LIN {X 0,Y 474.699,Z 291.349,A -85,B 0,C 180,E1 -7395.456,E2 -7395.456} C_VEL
LIN {X 0,Y 474.663,Z 291.357,A -85,B 0,C 180,E1 -7399.01,E2 -7399.01} C_VEL
LIN {X 0,Y 474.587,Z 291.362,A -85,B 0,C 180,E1 -7401.729,E2 -7401.729} C_VEL
LIN {X 0,Y 474.657,Z 291.358,A -85,B 0,C 180,E1 -7404.493,E2 -7404.493} C_VEL
LIN {X 0,Y 474.68,Z 291.352,A -85,B 0,C 180,E1 -7407.334,E2 -7407.334} C_VEL
LIN {X 0,Y 474.603,Z 291.361,A -85,B 0,C 180,E1 -7410.23,E2 -7410.23} C_VEL
LIN {X 0,Y 474.641,Z 291.362,A -85,B 0,C 180,E1 -7413.22,E2 -7413.22} C_VEL
LIN {X 0,Y 474.587,Z 291.364,A -85,B 0,C 180,E1 -7416.324,E2 -7416.324} C_VEL
LIN {X 0,Y 474.617,Z 291.362,A -85,B 0,C 180,E1 -7419.646,E2 -7419.646} C_VEL
LIN {X 0,Y 474.614,Z 291.363,A -85,B 0,C 180,E1 -7422.934,E2 -7422.934} C_VEL
LIN {X 0,Y 474.604,Z 291.365,A -85,B 0,C 180,E1 -7425.895,E2 -7425.895} C_VEL
LIN {X 0,Y 474.627,Z 291.361,A -85,B 0,C 180,E1 -7429.041,E2 -7429.041} C_VEL
LIN {X 0,Y 474.61,Z 291.365,A -85,B 0,C 180,E1 -7431.704,E2 -7431.704} C_VEL
LIN {X 0,Y 474.624,Z 291.359,A -85,B 0,C 180,E1 -7434.726,E2 -7434.726} C_VEL
LIN {X 0,Y 474.636,Z 291.366,A -85,B 0,C 180,E1 -7437.788,E2 -7437.788} C_VEL
LIN {X 0,Y 474.641,Z 291.389,A -85,B 0,C 180,E1 -7439.43,E2 -7439.43} C_VEL
LIN {X 0,Y 475.664,Z 297.352,A -85,B 0,C 180,E1 -7440.661,E2 -7440.661} C_VEL
LIN {X 0,Y 475.45,Z 310.857,A -85,B 0,C 180,E1 -7443.24,E2 -7443.24} C_VEL
LIN {X 0,Y 478.358,Z 325.969,A -85,B 0,C 180,E1 -7443.591,E2 -7443.591} C_VEL
LIN {X 0,Y 477.959,Z 363.89,A -85,B 0,C 180,E1 -7444.164,E2 -7444.164} C_VEL
LIN {X 0,Y 477.193,Z 369.733,A -85,B 0,C 180,E1 -7444.225,E2 -7444.225} C_VEL
LIN {X 0,Y 471.606,Z 388.747,A -85,B 0,C 180,E1 -7444.31,E2 -7444.31} C_VEL
LIN {X 0,Y 470.888,Z 394.589,A -85,B 0,C 180,E1 -7444.374,E2 -7444.374} C_VEL
LIN {X 0,Y 470.679,Z 419.305,A -85,B 0,C 180,E1 -7444.785,E2 -7444.785} C_VEL
LIN {X 0,Y 470.335,Z 432.586,A -85,B 0,C 180,E1 -7445.178,E2 -7445.178} C_VEL
LIN {X 0,Y 470.093,Z 444.455,A -85,B 0,C 180,E1 -7445.702,E2 -7445.702} C_VEL
LIN {X 0,Y 469.632,Z 456.314,A -85,B 0,C 180,E1 -7446.402,E2 -7446.402} C_VEL
LIN {X 0,Y 469.071,Z 468.144,A -85,B 0,C 180,E1 -7447.306,E2 -7447.306} C_VEL
LIN {X 0,Y 468.611,Z 478.255,A -85,B 0,C 180,E1 -7448.276,E2 -7448.276} C_VEL
LIN {X 0,Y 468.134,Z 487.264,A -85,B 0,C 180,E1 -7449.341,E2 -7449.341} C_VEL
LIN {X 0,Y 467.759,Z 495.099,A -85,B 0,C 180,E1 -7450.47,E2 -7450.47} C_VEL
LIN {X 0,Y 467.356,Z 502.71,A -85,B 0,C 180,E1 -7451.818,E2 -7451.818} C_VEL
LIN {X 0,Y 467.119,Z 507.836,A -85,B 0,C 180,E1 -7452.939,E2 -7452.939} C_VEL
LIN {X 0,Y 466.914,Z 513.267,A -85,B 0,C 180,E1 -7454.436,E2 -7454.436} C_VEL
LIN {X 0,Y 466.804,Z 516.504,A -85,B 0,C 180,E1 -7455.616,E2 -7455.616} C_VEL
LIN {X 0,Y 466.642,Z 519.178,A -85,B 0,C 180,E1 -7456.943,E2 -7456.943} C_VEL
LIN {X 0,Y 466.683,Z 520.801,A -85,B 0,C 180,E1 -7458.2,E2 -7458.2} C_VEL
LIN {X 0,Y 466.618,Z 521.619,A -85,B 0,C 180,E1 -7459.587,E2 -7459.587} C_VEL
LIN {X 0,Y 466.608,Z 521.219,A -85,B 0,C 180,E1 -7461.337,E2 -7461.337} C_VEL
LIN {X 0,Y 466.648,Z 520.4,A -85,B 0,C 180,E1 -7462.209,E2 -7462.209} C_VEL
LIN {X 0,Y 466.771,Z 518.274,A -85,B 0,C 180,E1 -7463.585,E2 -7463.585} C_VEL
LIN {X 0,Y 466.796,Z 515.477,A -85,B 0,C 180,E1 -7464.817,E2 -7464.817} C_VEL
LIN {X 0,Y 466.926,Z 511.505,A -85,B 0,C 180,E1 -7466.116,E2 -7466.116} C_VEL
LIN {X 0,Y 467.112,Z 505.404,A -85,B 0,C 180,E1 -7467.628,E2 -7467.628} C_VEL
LIN {X 0,Y 467.432,Z 498.758,A -85,B 0,C 180,E1 -7468.923,E2 -7468.923} C_VEL
LIN {X 0,Y 467.848,Z 490.53,A -85,B 0,C 180,E1 -7470.215,E2 -7470.215} C_VEL
LIN {X 0,Y 468.168,Z 482.104,A -85,B 0,C 180,E1 -7471.29,E2 -7471.29} C_VEL
LIN {X 0,Y 468.605,Z 471.721,A -85,B 0,C 180,E1 -7472.363,E2 -7472.363} C_VEL
LIN {X 0,Y 469.234,Z 461.395,A -85,B 0,C 180,E1 -7473.219,E2 -7473.219} C_VEL
LIN {X 0,Y 469.692,Z 450.127,A -85,B 0,C 180,E1 -7473.968,E2 -7473.968} C_VEL
LIN {X 0,Y 470.052,Z 438.556,A -85,B 0,C 180,E1 -7474.555,E2 -7474.555} C_VEL
LIN {X 0,Y 470.323,Z 426.176,A -85,B 0,C 180,E1 -7475.009,E2 -7475.009} C_VEL
LIN {X 0,Y 470.539,Z 413.632,A -85,B 0,C 180,E1 -7475.302,E2 -7475.302} C_VEL
LIN {X 0,Y 471.218,Z 325.536,A -85,B 0,C 180,E1 -7476.65,E2 -7476.65} C_VEL
LIN {X 0,Y 468.385,Z 310.756,A -85,B 0,C 180,E1 -7477.002,E2 -7477.002} C_VEL
LIN {X 0,Y 468.608,Z 299.276,A -85,B 0,C 180,E1 -7479.277,E2 -7479.277} C_VEL
LIN {X 0,Y 467.603,Z 292.239,A -85,B 0,C 180,E1 -7480.746,E2 -7480.746} C_VEL
LIN {X 0,Y 467.583,Z 292.239,A -85,B 0,C 180,E1 -7483.029,E2 -7483.029} C_VEL
LIN {X 0,Y 467.623,Z 292.233,A -85,B 0,C 180,E1 -7485.873,E2 -7485.873} C_VEL
LIN {X 0,Y 467.615,Z 292.231,A -85,B 0,C 180,E1 -7489.307,E2 -7489.307} C_VEL
LIN {X 0,Y 467.529,Z 292.245,A -85,B 0,C 180,E1 -7492.073,E2 -7492.073} C_VEL
LIN {X 0,Y 467.551,Z 292.244,A -85,B 0,C 180,E1 -7494.889,E2 -7494.889} C_VEL
LIN {X 0,Y 467.542,Z 292.241,A -85,B 0,C 180,E1 -7497.773,E2 -7497.773} C_VEL
LIN {X 0,Y 467.543,Z 292.245,A -85,B 0,C 180,E1 -7501.04,E2 -7501.04} C_VEL
LIN {X 0,Y 467.573,Z 292.238,A -85,B 0,C 180,E1 -7504.239,E2 -7504.239} C_VEL
LIN {X 0,Y 467.542,Z 292.245,A -85,B 0,C 180,E1 -7507.185,E2 -7507.185} C_VEL
LIN {X 0,Y 467.553,Z 292.24,A -85,B 0,C 180,E1 -7510.266,E2 -7510.266} C_VEL
LIN {X 0,Y 467.54,Z 292.242,A -85,B 0,C 180,E1 -7513.745,E2 -7513.745} C_VEL
LIN {X 0,Y 467.541,Z 292.241,A -85,B 0,C 180,E1 -7516.254,E2 -7516.254} C_VEL
LIN {X 0,Y 467.568,Z 292.24,A -85,B 0,C 180,E1 -7518.723,E2 -7518.723} C_VEL
LIN {X 0,Y 467.556,Z 292.24,A -85,B 0,C 180,E1 -7521.955,E2 -7521.955} C_VEL
LIN {X 0,Y 467.557,Z 292.244,A -85,B 0,C 180,E1 -7525.167,E2 -7525.167} C_VEL
LIN {X 0,Y 467.575,Z 292.237,A -85,B 0,C 180,E1 -7528.259,E2 -7528.259} C_VEL
LIN {X 0,Y 467.565,Z 292.242,A -85,B 0,C 180,E1 -7531.25,E2 -7531.25} C_VEL
LIN {X 0,Y 467.583,Z 292.237,A -85,B 0,C 180,E1 -7534.158,E2 -7534.158} C_VEL
LIN {X 0,Y 467.567,Z 292.238,A -85,B 0,C 180,E1 -7536.995,E2 -7536.995} C_VEL
LIN {X 0,Y 467.614,Z 292.241,A -85,B 0,C 180,E1 -7539.777,E2 -7539.777} C_VEL
LIN {X 0,Y 467.599,Z 292.234,A -85,B 0,C 180,E1 -7542.506,E2 -7542.506} C_VEL
LIN {X 0,Y 467.596,Z 292.234,A -85,B 0,C 180,E1 -7545.196,E2 -7545.196} C_VEL
LIN {X 0,Y 467.647,Z 292.234,A -85,B 0,C 180,E1 -7547.854,E2 -7547.854} C_VEL
LIN {X 0,Y 467.672,Z 292.225,A -85,B 0,C 180,E1 -7551.357,E2 -7551.357} C_VEL
LIN {X 0,Y 467.712,Z 292.225,A -85,B 0,C 180,E1 -7553.962,E2 -7553.962} C_VEL
LIN {X 0,Y 467.85,Z 292.202,A -85,B 0,C 180,E1 -7557.417,E2 -7557.417} C_VEL
LIN {X 0,Y 467.871,Z 292.204,A -85,B 0,C 180,E1 -7560,E2 -7560} C_VEL
LIN {X 0,Y 467.85,Z 292.208,A -85,B 0,C 180,E1 -7562.583,E2 -7562.583} C_VEL
LIN {X 0,Y 467.734,Z 292.219,A -85,B 0,C 180,E1 -7566.038,E2 -7566.038} C_VEL
LIN {X 0,Y 467.674,Z 292.232,A -85,B 0,C 180,E1 -7568.643,E2 -7568.643} C_VEL
LIN {X 0,Y 467.648,Z 292.23,A -85,B 0,C 180,E1 -7572.146,E2 -7572.146} C_VEL
LIN {X 0,Y 467.631,Z 292.229,A -85,B 0,C 180,E1 -7575.695,E2 -7575.695} C_VEL
LIN {X 0,Y 467.609,Z 292.241,A -85,B 0,C 180,E1 -7578.765,E2 -7578.765} C_VEL
LIN {X 0,Y 467.572,Z 292.24,A -85,B 0,C 180,E1 -7581.269,E2 -7581.269} C_VEL
LIN {X 0,Y 467.566,Z 292.238,A -85,B 0,C 180,E1 -7583.944,E2 -7583.944} C_VEL
LIN {X 0,Y 467.621,Z 292.236,A -85,B 0,C 180,E1 -7586.8,E2 -7586.8} C_VEL
LIN {X 0,Y 467.582,Z 292.237,A -85,B 0,C 180,E1 -7589.736,E2 -7589.736} C_VEL
LIN {X 0,Y 467.577,Z 292.239,A -85,B 0,C 180,E1 -7592.759,E2 -7592.759} C_VEL
LIN {X 0,Y 467.55,Z 292.241,A -85,B 0,C 180,E1 -7595.89,E2 -7595.89} C_VEL
LIN {X 0,Y 467.577,Z 292.242,A -85,B 0,C 180,E1 -7599.145,E2 -7599.145} C_VEL
LIN {X 0,Y 467.582,Z 292.236,A -85,B 0,C 180,E1 -7602.568,E2 -7602.568} C_VEL
LIN {X 0,Y 467.566,Z 292.24,A -85,B 0,C 180,E1 -7605.054,E2 -7605.054} C_VEL
LIN {X 0,Y 467.585,Z 292.242,A -85,B 0,C 180,E1 -7607.441,E2 -7607.441} C_VEL
LIN {X 0,Y 467.557,Z 292.239,A -85,B 0,C 180,E1 -7610.854,E2 -7610.854} C_VEL
LIN {X 0,Y 467.557,Z 292.241,A -85,B 0,C 180,E1 -7614.262,E2 -7614.262} C_VEL
LIN {X 0,Y 467.58,Z 292.238,A -85,B 0,C 180,E1 -7617.322,E2 -7617.322} C_VEL
LIN {X 0,Y 467.569,Z 292.241,A -85,B 0,C 180,E1 -7620.668,E2 -7620.668} C_VEL
LIN {X 0,Y 467.628,Z 292.238,A -85,B 0,C 180,E1 -7623.683,E2 -7623.683} C_VEL
LIN {X 0,Y 467.684,Z 292.443,A -85,B 0,C 180,E1 -7624.106,E2 -7624.106} C_VEL
LIN {X 0,Y 469.76,Z 303.592,A -85,B 0,C 180,E1 -7626.176,E2 -7626.176} C_VEL
LIN {X 0,Y 469.177,Z 319.502,A -85,B 0,C 180,E1 -7628.931,E2 -7628.931} C_VEL
LIN {X 0,Y 468.445,Z 337.977,A -85,B 0,C 180,E1 -7632.089,E2 -7632.089} C_VEL
LIN {X 0,Y 468.223,Z 343.562,A -85,B 0,C 180,E1 -7633.037,E2 -7633.037} C_VEL
LIN {X 0,Y 471.029,Z 362.98,A -85,B 0,C 180,E1 -7633.437,E2 -7633.437} C_VEL
LIN {X 0,Y 470.381,Z 452.058,A -85,B 0,C 180,E1 -7634.816,E2 -7634.816} C_VEL
LIN {X 0,Y 470.087,Z 465.35,A -85,B 0,C 180,E1 -7635.194,E2 -7635.194} C_VEL
LIN {X 0,Y 469.635,Z 477.531,A -85,B 0,C 180,E1 -7635.705,E2 -7635.705} C_VEL
LIN {X 0,Y 469.193,Z 489.014,A -85,B 0,C 180,E1 -7636.355,E2 -7636.355} C_VEL
LIN {X 0,Y 468.662,Z 501.141,A -85,B 0,C 180,E1 -7637.25,E2 -7637.25} C_VEL
LIN {X 0,Y 468.214,Z 511.384,A -85,B 0,C 180,E1 -7638.2,E2 -7638.2} C_VEL
LIN {X 0,Y 467.766,Z 520.021,A -85,B 0,C 180,E1 -7639.176,E2 -7639.176} C_VEL
LIN {X 0,Y 467.411,Z 527.986,A -85,B 0,C 180,E1 -7640.262,E2 -7640.262} C_VEL
LIN {X 0,Y 467.109,Z 535.769,A -85,B 0,C 180,E1 -7641.565,E2 -7641.565} C_VEL
LIN {X 0,Y 466.85,Z 542.921,A -85,B 0,C 180,E1 -7643.083,E2 -7643.083} C_VEL
LIN {X 0,Y 466.76,Z 547.684,A -85,B 0,C 180,E1 -7644.384,E2 -7644.384} C_VEL
LIN {X 0,Y 466.647,Z 551.321,A -85,B 0,C 180,E1 -7645.682,E2 -7645.682} C_VEL
LIN {X 0,Y 466.69,Z 553.202,A -85,B 0,C 180,E1 -7646.547,E2 -7646.547} C_VEL
LIN {X 0,Y 466.662,Z 554.611,A -85,B 0,C 180,E1 -7647.411,E2 -7647.411} C_VEL
LIN {X 0,Y 466.619,Z 556.227,A -85,B 0,C 180,E1 -7649.137,E2 -7649.137} C_VEL
LIN {X 0,Y 466.601,Z 556.45,A -85,B 0,C 180,E1 -7650,E2 -7650} C_VEL
LIN {X 0,Y 466.619,Z 556.241,A -85,B 0,C 180,E1 -7650.863,E2 -7650.863} C_VEL
LIN {X 0,Y 466.662,Z 554.643,A -85,B 0,C 180,E1 -7652.59,E2 -7652.59} C_VEL
LIN {X 0,Y 466.69,Z 553.251,A -85,B 0,C 180,E1 -7653.454,E2 -7653.454} C_VEL
LIN {X 0,Y 466.689,Z 550.317,A -85,B 0,C 180,E1 -7654.751,E2 -7654.751} C_VEL
LIN {X 0,Y 466.751,Z 546.351,A -85,B 0,C 180,E1 -7656.051,E2 -7656.051} C_VEL
LIN {X 0,Y 466.943,Z 540.263,A -85,B 0,C 180,E1 -7657.568,E2 -7657.568} C_VEL
LIN {X 0,Y 467.186,Z 533.607,A -85,B 0,C 180,E1 -7658.87,E2 -7658.87} C_VEL
LIN {X 0,Y 467.537,Z 525.357,A -85,B 0,C 180,E1 -7660.174,E2 -7660.174} C_VEL
LIN {X 0,Y 468.026,Z 516.93,A -85,B 0,C 180,E1 -7661.257,E2 -7661.257} C_VEL
LIN {X 0,Y 468.529,Z 506.943,A -85,B 0,C 180,E1 -7662.305,E2 -7662.305} C_VEL
LIN {X 0,Y 468.957,Z 496.271,A -85,B 0,C 180,E1 -7663.212,E2 -7663.212} C_VEL
LIN {X 0,Y 469.489,Z 485.054,A -85,B 0,C 180,E1 -7663.968,E2 -7663.968} C_VEL
LIN {X 0,Y 469.977,Z 473.698,A -85,B 0,C 180,E1 -7664.561,E2 -7664.561} C_VEL
LIN {X 0,Y 470.38,Z 460.827,A -85,B 0,C 180,E1 -7665.047,E2 -7665.047} C_VEL
LIN {X 0,Y 470.681,Z 447.177,A -85,B 0,C 180,E1 -7665.369,E2 -7665.369} C_VEL
LIN {X 0,Y 471.268,Z 361.934,A -85,B 0,C 180,E1 -7666.688,E2 -7666.688} C_VEL
LIN {X 0,Y 468.32,Z 343.326,A -85,B 0,C 180,E1 -7667.112,E2 -7667.112} C_VEL
LIN {X 0,Y 469.089,Z 325.621,A -85,B 0,C 180,E1 -7670.157,E2 -7670.157} C_VEL
LIN {X 0,Y 469.915,Z 307.359,A -85,B 0,C 180,E1 -7673.349,E2 -7673.349} C_VEL
LIN {X 0,Y 469.787,Z 302.998,A -85,B 0,C 180,E1 -7674.138,E2 -7674.138} C_VEL
LIN {X 0,Y 467.646,Z 292.237,A -85,B 0,C 180,E1 -7676.257,E2 -7676.257} C_VEL
LIN {X 0,Y 467.572,Z 292.244,A -85,B 0,C 180,E1 -7679.332,E2 -7679.332} C_VEL
LIN {X 0,Y 467.584,Z 292.238,A -85,B 0,C 180,E1 -7682.679,E2 -7682.679} C_VEL
LIN {X 0,Y 467.561,Z 292.242,A -85,B 0,C 180,E1 -7685.739,E2 -7685.739} C_VEL
LIN {X 0,Y 467.561,Z 292.241,A -85,B 0,C 180,E1 -7689.147,E2 -7689.147} C_VEL
LIN {X 0,Y 467.588,Z 292.242,A -85,B 0,C 180,E1 -7692.567,E2 -7692.567} C_VEL
LIN {X 0,Y 467.566,Z 292.242,A -85,B 0,C 180,E1 -7695.052,E2 -7695.052} C_VEL
LIN {X 0,Y 467.59,Z 292.235,A -85,B 0,C 180,E1 -7697.44,E2 -7697.44} C_VEL
LIN {X 0,Y 467.576,Z 292.245,A -85,B 0,C 180,E1 -7700.854,E2 -7700.854} C_VEL
LIN {X 0,Y 467.559,Z 292.24,A -85,B 0,C 180,E1 -7704.261,E2 -7704.261} C_VEL
LIN {X 0,Y 467.581,Z 292.24,A -85,B 0,C 180,E1 -7707.321,E2 -7707.321} C_VEL
LIN {X 0,Y 467.569,Z 292.239,A -85,B 0,C 180,E1 -7710.667,E2 -7710.667} C_VEL
LIN {X 0,Y 467.615,Z 292.237,A -85,B 0,C 180,E1 -7713.199,E2 -7713.199} C_VEL
LIN {X 0,Y 467.592,Z 292.235,A -85,B 0,C 180,E1 -7716.468,E2 -7716.468} C_VEL
LIN {X 0,Y 467.621,Z 292.233,A -85,B 0,C 180,E1 -7719.777,E2 -7719.777} C_VEL
LIN {X 0,Y 467.607,Z 292.231,A -85,B 0,C 180,E1 -7722.507,E2 -7722.507} C_VEL
LIN {X 0,Y 467.608,Z 292.235,A -85,B 0,C 180,E1 -7725.196,E2 -7725.196} C_VEL
LIN {X 0,Y 467.654,Z 292.231,A -85,B 0,C 180,E1 -7727.854,E2 -7727.854} C_VEL
LIN {X 0,Y 467.68,Z 292.224,A -85,B 0,C 180,E1 -7731.357,E2 -7731.357} C_VEL
LIN {X 0,Y 467.741,Z 292.217,A -85,B 0,C 180,E1 -7733.962,E2 -7733.962} C_VEL
LIN {X 0,Y 467.858,Z 292.202,A -85,B 0,C 180,E1 -7737.417,E2 -7737.417} C_VEL
LIN {X 0,Y 467.88,Z 292.201,A -85,B 0,C 180,E1 -7740,E2 -7740} C_VEL
LIN {X 0,Y 467.857,Z 292.199,A -85,B 0,C 180,E1 -7742.583,E2 -7742.583} C_VEL
LIN {X 0,Y 467.732,Z 292.222,A -85,B 0,C 180,E1 -7746.037,E2 -7746.037} C_VEL
LIN {X 0,Y 467.679,Z 292.226,A -85,B 0,C 180,E1 -7748.643,E2 -7748.643} C_VEL
LIN {X 0,Y 467.654,Z 292.23,A -85,B 0,C 180,E1 -7752.145,E2 -7752.145} C_VEL
LIN {X 0,Y 467.638,Z 292.228,A -85,B 0,C 180,E1 -7755.695,E2 -7755.695} C_VEL
LIN {X 0,Y 467.616,Z 292.238,A -85,B 0,C 180,E1 -7758.764,E2 -7758.764} C_VEL
LIN {X 0,Y 467.579,Z 292.237,A -85,B 0,C 180,E1 -7761.268,E2 -7761.268} C_VEL
LIN {X 0,Y 467.571,Z 292.237,A -85,B 0,C 180,E1 -7763.943,E2 -7763.943} C_VEL
LIN {X 0,Y 467.616,Z 292.239,A -85,B 0,C 180,E1 -7766.8,E2 -7766.8} C_VEL
LIN {X 0,Y 467.552,Z 292.239,A -85,B 0,C 180,E1 -7769.738,E2 -7769.738} C_VEL
LIN {X 0,Y 467.582,Z 292.238,A -85,B 0,C 180,E1 -7772.758,E2 -7772.758} C_VEL
LIN {X 0,Y 467.552,Z 292.24,A -85,B 0,C 180,E1 -7775.89,E2 -7775.89} C_VEL
LIN {X 0,Y 467.575,Z 292.244,A -85,B 0,C 180,E1 -7779.145,E2 -7779.145} C_VEL
LIN {X 0,Y 467.586,Z 292.236,A -85,B 0,C 180,E1 -7782.567,E2 -7782.567} C_VEL
LIN {X 0,Y 467.565,Z 292.242,A -85,B 0,C 180,E1 -7785.053,E2 -7785.053} C_VEL
LIN {X 0,Y 467.589,Z 292.243,A -85,B 0,C 180,E1 -7787.44,E2 -7787.44} C_VEL
LIN {X 0,Y 467.56,Z 292.242,A -85,B 0,C 180,E1 -7790.853,E2 -7790.853} C_VEL
LIN {X 0,Y 467.56,Z 292.241,A -85,B 0,C 180,E1 -7794.261,E2 -7794.261} C_VEL
LIN {X 0,Y 467.582,Z 292.242,A -85,B 0,C 180,E1 -7797.321,E2 -7797.321} C_VEL
LIN {X 0,Y 467.594,Z 292.36,A -85,B 0,C 180,E1 -7799.239,E2 -7799.239} C_VEL
LIN {X 0,Y 468.745,Z 298.656,A -85,B 0,C 180,E1 -7800.557,E2 -7800.557} C_VEL
LIN {X 0,Y 468.479,Z 310.772,A -85,B 0,C 180,E1 -7802.933,E2 -7802.933} C_VEL
LIN {X 0,Y 471.552,Z 325.879,A -85,B 0,C 180,E1 -7803.319,E2 -7803.319} C_VEL
LIN {X 0,Y 470.888,Z 394.589,A -85,B 0,C 180,E1 -7804.374,E2 -7804.374} C_VEL
LIN {X 0,Y 470.185,Z 400.44,A -85,B 0,C 180,E1 -7804.435,E2 -7804.435} C_VEL
LIN {X 0,Y 464.632,Z 419.436,A -85,B 0,C 180,E1 -7804.553,E2 -7804.553} C_VEL
LIN {X 0,Y 463.798,Z 425.188,A -85,B 0,C 180,E1 -7804.679,E2 -7804.679} C_VEL
LIN {X 0,Y 463.444,Z 437.893,A -85,B 0,C 180,E1 -7805.138,E2 -7805.138} C_VEL
LIN {X 0,Y 463.017,Z 450.879,A -85,B 0,C 180,E1 -7805.806,E2 -7805.806} C_VEL
LIN {X 0,Y 462.522,Z 462.577,A -85,B 0,C 180,E1 -7806.611,E2 -7806.611} C_VEL
LIN {X 0,Y 461.987,Z 473.16,A -85,B 0,C 180,E1 -7807.529,E2 -7807.529} C_VEL
LIN {X 0,Y 461.451,Z 482.796,A -85,B 0,C 180,E1 -7808.56,E2 -7808.56} C_VEL
LIN {X 0,Y 460.975,Z 491.478,A -85,B 0,C 180,E1 -7809.705,E2 -7809.705} C_VEL
LIN {X 0,Y 460.513,Z 500.117,A -85,B 0,C 180,E1 -7811.12,E2 -7811.12} C_VEL
LIN {X 0,Y 460.2,Z 505.551,A -85,B 0,C 180,E1 -7812.216,E2 -7812.216} C_VEL
LIN {X 0,Y 459.96,Z 511.041,A -85,B 0,C 180,E1 -7813.58,E2 -7813.58} C_VEL
LIN {X 0,Y 459.776,Z 515.282,A -85,B 0,C 180,E1 -7814.938,E2 -7814.938} C_VEL
LIN {X 0,Y 459.663,Z 517.502,A -85,B 0,C 180,E1 -7815.84,E2 -7815.84} C_VEL
LIN {X 0,Y 459.579,Z 519.218,A -85,B 0,C 180,E1 -7816.739,E2 -7816.739} C_VEL
LIN {X 0,Y 459.589,Z 521.062,A -85,B 0,C 180,E1 -7818.148,E2 -7818.148} C_VEL
LIN {X 0,Y 459.537,Z 521.859,A -85,B 0,C 180,E1 -7819.425,E2 -7819.425} C_VEL
LIN {X 0,Y 459.504,Z 521.559,A -85,B 0,C 180,E1 -7821.202,E2 -7821.202} C_VEL
LIN {X 0,Y 459.543,Z 520.826,A -85,B 0,C 180,E1 -7822.088,E2 -7822.088} C_VEL
LIN {X 0,Y 459.694,Z 518.602,A -85,B 0,C 180,E1 -7823.589,E2 -7823.589} C_VEL
LIN {X 0,Y 459.7,Z 514.895,A -85,B 0,C 180,E1 -7825.176,E2 -7825.176} C_VEL
LIN {X 0,Y 459.897,Z 510.664,A -85,B 0,C 180,E1 -7826.495,E2 -7826.495} C_VEL
LIN {X 0,Y 460.144,Z 504.274,A -85,B 0,C 180,E1 -7828.03,E2 -7828.03} C_VEL
LIN {X 0,Y 460.532,Z 497.276,A -85,B 0,C 180,E1 -7829.344,E2 -7829.344} C_VEL
LIN {X 0,Y 460.953,Z 488.565,A -85,B 0,C 180,E1 -7830.655,E2 -7830.655} C_VEL
LIN {X 0,Y 461.333,Z 479.669,A -85,B 0,C 180,E1 -7831.745,E2 -7831.745} C_VEL
LIN {X 0,Y 461.819,Z 469.877,A -85,B 0,C 180,E1 -7832.725,E2 -7832.725} C_VEL
LIN {X 0,Y 462.457,Z 458.993,A -85,B 0,C 180,E1 -7833.594,E2 -7833.594} C_VEL
LIN {X 0,Y 462.878,Z 446.893,A -85,B 0,C 180,E1 -7834.353,E2 -7834.353} C_VEL
LIN {X 0,Y 463.252,Z 434.164,A -85,B 0,C 180,E1 -7834.949,E2 -7834.949} C_VEL
LIN {X 0,Y 463.548,Z 424.373,A -85,B 0,C 180,E1 -7835.273,E2 -7835.273} C_VEL
LIN {X 0,Y 463.692,Z 411.98,A -85,B 0,C 180,E1 -7835.544,E2 -7835.544} C_VEL
LIN {X 0,Y 464.345,Z 326.215,A -85,B 0,C 180,E1 -7836.873,E2 -7836.873} C_VEL
LIN {X 0,Y 461.404,Z 311.097,A -85,B 0,C 180,E1 -7837.218,E2 -7837.218} C_VEL
LIN {X 0,Y 461.623,Z 300.107,A -85,B 0,C 180,E1 -7839.419,E2 -7839.419} C_VEL
LIN {X 0,Y 460.573,Z 293.114,A -85,B 0,C 180,E1 -7840.912,E2 -7840.912} C_VEL
LIN {X 0,Y 460.537,Z 293.116,A -85,B 0,C 180,E1 -7843.232,E2 -7843.232} C_VEL
LIN {X 0,Y 460.578,Z 293.112,A -85,B 0,C 180,E1 -7845.987,E2 -7845.987} C_VEL
LIN {X 0,Y 460.562,Z 293.11,A -85,B 0,C 180,E1 -7849.615,E2 -7849.615} C_VEL
LIN {X 0,Y 460.505,Z 293.125,A -85,B 0,C 180,E1 -7852.428,E2 -7852.428} C_VEL
LIN {X 0,Y 460.529,Z 293.114,A -85,B 0,C 180,E1 -7855.792,E2 -7855.792} C_VEL
LIN {X 0,Y 460.516,Z 293.118,A -85,B 0,C 180,E1 -7859.232,E2 -7859.232} C_VEL
LIN {X 0,Y 460.525,Z 293.117,A -85,B 0,C 180,E1 -7862.284,E2 -7862.284} C_VEL
LIN {X 0,Y 460.504,Z 293.119,A -85,B 0,C 180,E1 -7865.445,E2 -7865.445} C_VEL
LIN {X 0,Y 460.524,Z 293.123,A -85,B 0,C 180,E1 -7868.894,E2 -7868.894} C_VEL
LIN {X 0,Y 460.485,Z 293.12,A -85,B 0,C 180,E1 -7872.184,E2 -7872.184} C_VEL
LIN {X 0,Y 460.506,Z 293.122,A -85,B 0,C 180,E1 -7875.41,E2 -7875.41} C_VEL
LIN {X 0,Y 460.52,Z 293.121,A -85,B 0,C 180,E1 -7878.988,E2 -7878.988} C_VEL
LIN {X 0,Y 460.508,Z 293.126,A -85,B 0,C 180,E1 -7881.265,E2 -7881.265} C_VEL
LIN {X 0,Y 460.503,Z 293.118,A -85,B 0,C 180,E1 -7884.554,E2 -7884.554} C_VEL
LIN {X 0,Y 460.523,Z 293.12,A -85,B 0,C 180,E1 -7887.715,E2 -7887.715} C_VEL
LIN {X 0,Y 460.529,Z 293.115,A -85,B 0,C 180,E1 -7890.768,E2 -7890.768} C_VEL
LIN {X 0,Y 460.537,Z 293.12,A -85,B 0,C 180,E1 -7893.733,E2 -7893.733} C_VEL
LIN {X 0,Y 460.536,Z 293.113,A -85,B 0,C 180,E1 -7896.623,E2 -7896.623} C_VEL
LIN {X 0,Y 460.542,Z 293.117,A -85,B 0,C 180,E1 -7899.452,E2 -7899.452} C_VEL
LIN {X 0,Y 460.55,Z 293.115,A -85,B 0,C 180,E1 -7902.23,E2 -7902.23} C_VEL
LIN {X 0,Y 460.559,Z 293.11,A -85,B 0,C 180,E1 -7904.965,E2 -7904.965} C_VEL
LIN {X 0,Y 460.602,Z 293.107,A -85,B 0,C 180,E1 -7908.559,E2 -7908.559} C_VEL
LIN {X 0,Y 460.657,Z 293.107,A -85,B 0,C 180,E1 -7912.108,E2 -7912.108} C_VEL
LIN {X 0,Y 460.681,Z 293.097,A -85,B 0,C 180,E1 -7914.748,E2 -7914.748} C_VEL
LIN {X 0,Y 460.792,Z 293.082,A -85,B 0,C 180,E1 -7917.378,E2 -7917.378} C_VEL
LIN {X 0,Y 460.842,Z 293.079,A -85,B 0,C 180,E1 -7920,E2 -7920} C_VEL
LIN {X 0,Y 460.791,Z 293.087,A -85,B 0,C 180,E1 -7922.623,E2 -7922.623} C_VEL
LIN {X 0,Y 460.701,Z 293.097,A -85,B 0,C 180,E1 -7926.13,E2 -7926.13} C_VEL
LIN {X 0,Y 460.621,Z 293.108,A -85,B 0,C 180,E1 -7928.776,E2 -7928.776} C_VEL
LIN {X 0,Y 460.605,Z 293.111,A -85,B 0,C 180,E1 -7932.445,E2 -7932.445} C_VEL
LIN {X 0,Y 460.592,Z 293.107,A -85,B 0,C 180,E1 -7935.998,E2 -7935.998} C_VEL
LIN {X 0,Y 460.563,Z 293.118,A -85,B 0,C 180,E1 -7938.902,E2 -7938.902} C_VEL
LIN {X 0,Y 460.508,Z 293.118,A -85,B 0,C 180,E1 -7941.486,E2 -7941.486} C_VEL
LIN {X 0,Y 460.535,Z 293.115,A -85,B 0,C 180,E1 -7944.333,E2 -7944.333} C_VEL
LIN {X 0,Y 460.578,Z 293.114,A -85,B 0,C 180,E1 -7947.244,E2 -7947.244} C_VEL
LIN {X 0,Y 460.524,Z 293.115,A -85,B 0,C 180,E1 -7950.239,E2 -7950.239} C_VEL
LIN {X 0,Y 460.523,Z 293.122,A -85,B 0,C 180,E1 -7953.326,E2 -7953.326} C_VEL
LIN {X 0,Y 460.473,Z 293.122,A -85,B 0,C 180,E1 -7956.53,E2 -7956.53} C_VEL
LIN {X 0,Y 460.553,Z 293.114,A -85,B 0,C 180,E1 -7959.86,E2 -7959.86} C_VEL
LIN {X 0,Y 460.512,Z 293.118,A -85,B 0,C 180,E1 -7962.902,E2 -7962.902} C_VEL
LIN {X 0,Y 460.507,Z 293.121,A -85,B 0,C 180,E1 -7965.831,E2 -7965.831} C_VEL
LIN {X 0,Y 460.527,Z 293.116,A -85,B 0,C 180,E1 -7968.99,E2 -7968.99} C_VEL
LIN {X 0,Y 460.515,Z 293.119,A -85,B 0,C 180,E1 -7971.267,E2 -7971.267} C_VEL
LIN {X 0,Y 460.508,Z 293.117,A -85,B 0,C 180,E1 -7974.555,E2 -7974.555} C_VEL
LIN {X 0,Y 460.53,Z 293.121,A -85,B 0,C 180,E1 -7977.717,E2 -7977.717} C_VEL
LIN {X 0,Y 460.539,Z 293.117,A -85,B 0,C 180,E1 -7980.77,E2 -7980.77} C_VEL
LIN {X 0,Y 460.608,Z 293.165,A -85,B 0,C 180,E1 -7983.897,E2 -7983.897} C_VEL
LIN {X 0,Y 462.732,Z 304.47,A -85,B 0,C 180,E1 -7986.03,E2 -7986.03} C_VEL
LIN {X 0,Y 462.372,Z 315.661,A -85,B 0,C 180,E1 -7988.002,E2 -7988.002} C_VEL
LIN {X 0,Y 461.625,Z 334.927,A -85,B 0,C 180,E1 -7991.355,E2 -7991.355} C_VEL
LIN {X 0,Y 461.209,Z 343.319,A -85,B 0,C 180,E1 -7992.801,E2 -7992.801} C_VEL
LIN {X 0,Y 464.194,Z 363.447,A -85,B 0,C 180,E1 -7993.22,E2 -7993.22} C_VEL
LIN {X 0,Y 463.482,Z 452.039,A -85,B 0,C 180,E1 -7994.612,E2 -7994.612} C_VEL
LIN {X 0,Y 463.152,Z 465.254,A -85,B 0,C 180,E1 -7994.995,E2 -7994.995} C_VEL
LIN {X 0,Y 462.698,Z 477.97,A -85,B 0,C 180,E1 -7995.543,E2 -7995.543} C_VEL
LIN {X 0,Y 462.182,Z 490.059,A -85,B 0,C 180,E1 -7996.256,E2 -7996.256} C_VEL
LIN {X 0,Y 461.659,Z 501.639,A -85,B 0,C 180,E1 -7997.14,E2 -7997.14} C_VEL
LIN {X 0,Y 461.178,Z 512.005,A -85,B 0,C 180,E1 -7998.128,E2 -7998.128} C_VEL
LIN {X 0,Y 460.665,Z 521.329,A -85,B 0,C 180,E1 -7999.229,E2 -7999.229} C_VEL
LIN {X 0,Y 460.227,Z 530.378,A -85,B 0,C 180,E1 -8000.552,E2 -8000.552} C_VEL
LIN {X 0,Y 459.941,Z 537.666,A -85,B 0,C 180,E1 -8001.875,E2 -8001.875} C_VEL
LIN {X 0,Y 459.727,Z 543.86,A -85,B 0,C 180,E1 -8003.295,E2 -8003.295} C_VEL
LIN {X 0,Y 459.65,Z 548.701,A -85,B 0,C 180,E1 -8004.737,E2 -8004.737} C_VEL
LIN {X 0,Y 459.564,Z 551.018,A -85,B 0,C 180,E1 -8005.615,E2 -8005.615} C_VEL
LIN {X 0,Y 459.586,Z 552.907,A -85,B 0,C 180,E1 -8006.494,E2 -8006.494} C_VEL
LIN {X 0,Y 459.584,Z 554.328,A -85,B 0,C 180,E1 -8007.371,E2 -8007.371} C_VEL
LIN {X 0,Y 459.552,Z 555.956,A -85,B 0,C 180,E1 -8009.124,E2 -8009.124} C_VEL
LIN {X 0,Y 459.532,Z 556.186,A -85,B 0,C 180,E1 -8010,E2 -8010} C_VEL
LIN {X 0,Y 459.523,Z 555.985,A -85,B 0,C 180,E1 -8010.877,E2 -8010.877} C_VEL
LIN {X 0,Y 459.584,Z 554.398,A -85,B 0,C 180,E1 -8012.63,E2 -8012.63} C_VEL
LIN {X 0,Y 459.585,Z 553.013,A -85,B 0,C 180,E1 -8013.507,E2 -8013.507} C_VEL
LIN {X 0,Y 459.617,Z 550.091,A -85,B 0,C 180,E1 -8014.825,E2 -8014.825} C_VEL
LIN {X 0,Y 459.715,Z 545.124,A -85,B 0,C 180,E1 -8016.431,E2 -8016.431} C_VEL
LIN {X 0,Y 459.903,Z 539.062,A -85,B 0,C 180,E1 -8017.905,E2 -8017.905} C_VEL
LIN {X 0,Y 460.187,Z 532.203,A -85,B 0,C 180,E1 -8019.228,E2 -8019.228} C_VEL
LIN {X 0,Y 460.588,Z 523.666,A -85,B 0,C 180,E1 -8020.551,E2 -8020.551} C_VEL
LIN {X 0,Y 461.113,Z 514.906,A -85,B 0,C 180,E1 -8021.651,E2 -8021.651} C_VEL
LIN {X 0,Y 461.689,Z 504.044,A -85,B 0,C 180,E1 -8022.761,E2 -8022.761} C_VEL
LIN {X 0,Y 462.184,Z 493.401,A -85,B 0,C 180,E1 -8023.633,E2 -8023.633} C_VEL
LIN {X 0,Y 462.757,Z 481.363,A -85,B 0,C 180,E1 -8024.4,E2 -8024.4} C_VEL
LIN {X 0,Y 463.308,Z 468.832,A -85,B 0,C 180,E1 -8025.001,E2 -8025.001} C_VEL
LIN {X 0,Y 463.699,Z 456.735,A -85,B 0,C 180,E1 -8025.409,E2 -8025.409} C_VEL
LIN {X 0,Y 463.973,Z 441.511,A -85,B 0,C 180,E1 -8025.71,E2 -8025.71} C_VEL
LIN {X 0,Y 464.561,Z 363.362,A -85,B 0,C 180,E1 -8026.934,E2 -8026.934} C_VEL
LIN {X 0,Y 461.375,Z 343.091,A -85,B 0,C 180,E1 -8027.398,E2 -8027.398} C_VEL
LIN {X 0,Y 462.172,Z 325.515,A -85,B 0,C 180,E1 -8030.472,E2 -8030.472} C_VEL
LIN {X 0,Y 463.001,Z 308.573,A -85,B 0,C 180,E1 -8033.482,E2 -8033.482} C_VEL
LIN {X 0,Y 462.79,Z 303.974,A -85,B 0,C 180,E1 -8034.332,E2 -8034.332} C_VEL
LIN {X 0,Y 460.593,Z 293.115,A -85,B 0,C 180,E1 -8036.508,E2 -8036.508} C_VEL
LIN {X 0,Y 460.533,Z 293.123,A -85,B 0,C 180,E1 -8039.558,E2 -8039.558} C_VEL
LIN {X 0,Y 460.533,Z 293.12,A -85,B 0,C 180,E1 -8042.284,E2 -8042.284} C_VEL
LIN {X 0,Y 460.512,Z 293.119,A -85,B 0,C 180,E1 -8045.445,E2 -8045.445} C_VEL
LIN {X 0,Y 460.535,Z 293.118,A -85,B 0,C 180,E1 -8048.896,E2 -8048.896} C_VEL
LIN {X 0,Y 460.524,Z 293.121,A -85,B 0,C 180,E1 -8052.181,E2 -8052.181} C_VEL
LIN {X 0,Y 460.514,Z 293.118,A -85,B 0,C 180,E1 -8055.411,E2 -8055.411} C_VEL
LIN {X 0,Y 460.532,Z 293.119,A -85,B 0,C 180,E1 -8058.397,E2 -8058.397} C_VEL
LIN {X 0,Y 460.523,Z 293.118,A -85,B 0,C 180,E1 -8061.266,E2 -8061.266} C_VEL
LIN {X 0,Y 460.51,Z 293.121,A -85,B 0,C 180,E1 -8064.554,E2 -8064.554} C_VEL
LIN {X 0,Y 460.531,Z 293.115,A -85,B 0,C 180,E1 -8067.715,E2 -8067.715} C_VEL
LIN {X 0,Y 460.539,Z 293.116,A -85,B 0,C 180,E1 -8070.769,E2 -8070.769} C_VEL
LIN {X 0,Y 460.558,Z 293.112,A -85,B 0,C 180,E1 -8073.734,E2 -8073.734} C_VEL
LIN {X 0,Y 460.545,Z 293.113,A -85,B 0,C 180,E1 -8076.624,E2 -8076.624} C_VEL
LIN {X 0,Y 460.551,Z 293.119,A -85,B 0,C 180,E1 -8079.453,E2 -8079.453} C_VEL
LIN {X 0,Y 460.558,Z 293.11,A -85,B 0,C 180,E1 -8082.23,E2 -8082.23} C_VEL
LIN {X 0,Y 460.566,Z 293.11,A -85,B 0,C 180,E1 -8084.965,E2 -8084.965} C_VEL
LIN {X 0,Y 460.609,Z 293.103,A -85,B 0,C 180,E1 -8088.559,E2 -8088.559} C_VEL
LIN {X 0,Y 460.694,Z 293.096,A -85,B 0,C 180,E1 -8092.108,E2 -8092.108} C_VEL
LIN {X 0,Y 460.694,Z 293.088,A -85,B 0,C 180,E1 -8094.748,E2 -8094.748} C_VEL
LIN {X 0,Y 460.799,Z 293.081,A -85,B 0,C 180,E1 -8097.377,E2 -8097.377} C_VEL
LIN {X 0,Y 460.85,Z 293.077,A -85,B 0,C 180,E1 -8100,E2 -8100} C_VEL
LIN {X 0,Y 460.798,Z 293.078,A -85,B 0,C 180,E1 -8102.622,E2 -8102.622} C_VEL
LIN {X 0,Y 460.699,Z 293.1,A -85,B 0,C 180,E1 -8106.13,E2 -8106.13} C_VEL
LIN {X 0,Y 460.626,Z 293.103,A -85,B 0,C 180,E1 -8108.776,E2 -8108.776} C_VEL
LIN {X 0,Y 460.612,Z 293.107,A -85,B 0,C 180,E1 -8112.445,E2 -8112.445} C_VEL
LIN {X 0,Y 460.599,Z 293.107,A -85,B 0,C 180,E1 -8115.998,E2 -8115.998} C_VEL
LIN {X 0,Y 460.569,Z 293.114,A -85,B 0,C 180,E1 -8118.902,E2 -8118.902} C_VEL
LIN {X 0,Y 460.514,Z 293.116,A -85,B 0,C 180,E1 -8121.486,E2 -8121.486} C_VEL
LIN {X 0,Y 460.541,Z 293.115,A -85,B 0,C 180,E1 -8124.332,E2 -8124.332} C_VEL
LIN {X 0,Y 460.572,Z 293.11,A -85,B 0,C 180,E1 -8127.244,E2 -8127.244} C_VEL
LIN {X 0,Y 460.509,Z 293.117,A -85,B 0,C 180,E1 -8130.24,E2 -8130.24} C_VEL
LIN {X 0,Y 460.528,Z 293.118,A -85,B 0,C 180,E1 -8133.325,E2 -8133.325} C_VEL
LIN {X 0,Y 460.475,Z 293.123,A -85,B 0,C 180,E1 -8136.53,E2 -8136.53} C_VEL
LIN {X 0,Y 460.526,Z 293.115,A -85,B 0,C 180,E1 -8139.863,E2 -8139.863} C_VEL
LIN {X 0,Y 460.512,Z 293.12,A -85,B 0,C 180,E1 -8142.9,E2 -8142.9} C_VEL
LIN {X 0,Y 460.506,Z 293.122,A -85,B 0,C 180,E1 -8145.831,E2 -8145.831} C_VEL
LIN {X 0,Y 460.53,Z 293.117,A -85,B 0,C 180,E1 -8148.989,E2 -8148.989} C_VEL
LIN {X 0,Y 460.519,Z 293.122,A -85,B 0,C 180,E1 -8151.266,E2 -8151.266} C_VEL
LIN {X 0,Y 460.51,Z 293.118,A -85,B 0,C 180,E1 -8154.554,E2 -8154.554} C_VEL
LIN {X 0,Y 460.533,Z 293.122,A -85,B 0,C 180,E1 -8157.716,E2 -8157.716} C_VEL
LIN {X 0,Y 460.541,Z 293.173,A -85,B 0,C 180,E1 -8159,E2 -8159} C_VEL
LIN {X 0,Y 461.833,Z 300.406,A -85,B 0,C 180,E1 -8160.534,E2 -8160.534} C_VEL
LIN {X 0,Y 461.587,Z 311.081,A -85,B 0,C 180,E1 -8162.653,E2 -8162.653} C_VEL
LIN {X 0,Y 464.85,Z 327.03,A -85,B 0,C 180,E1 -8163.058,E2 -8163.058} C_VEL
LIN {X 0,Y 463.919,Z 418.723,A -85,B 0,C 180,E1 -8164.511,E2 -8164.511} C_VEL
LIN {X 0,Y 463.798,Z 425.188,A -85,B 0,C 180,E1 -8164.679,E2 -8164.679} C_VEL
LIN {X 0,Y 462.337,Z 432.771,A -85,B 0,C 180,E1 -8164.881,E2 -8164.881} C_VEL
LIN {X 0,Y 459.73,Z 440.103,A -85,B 0,C 180,E1 -8165.093,E2 -8165.093} C_VEL
LIN {X 0,Y 456.85,Z 449.124,A -85,B 0,C 180,E1 -8165.465,E2 -8165.465} C_VEL
LIN {X 0,Y 456.093,Z 454.379,A -85,B 0,C 180,E1 -8165.769,E2 -8165.769} C_VEL
LIN {X 0,Y 455.524,Z 465.525,A -85,B 0,C 180,E1 -8166.592,E2 -8166.592} C_VEL
LIN {X 0,Y 454.904,Z 476.454,A -85,B 0,C 180,E1 -8167.618,E2 -8167.618} C_VEL
LIN {X 0,Y 454.357,Z 485.667,A -85,B 0,C 180,E1 -8168.685,E2 -8168.685} C_VEL
LIN {X 0,Y 453.9,Z 493.899,A -85,B 0,C 180,E1 -8169.848,E2 -8169.848} C_VEL
LIN {X 0,Y 453.399,Z 501.867,A -85,B 0,C 180,E1 -8171.238,E2 -8171.238} C_VEL
LIN {X 0,Y 453.119,Z 507.252,A -85,B 0,C 180,E1 -8172.395,E2 -8172.395} C_VEL
LIN {X 0,Y 452.849,Z 512.415,A -85,B 0,C 180,E1 -8173.778,E2 -8173.778} C_VEL
LIN {X 0,Y 452.681,Z 516.379,A -85,B 0,C 180,E1 -8175.157,E2 -8175.157} C_VEL
LIN {X 0,Y 452.502,Z 519.263,A -85,B 0,C 180,E1 -8176.528,E2 -8176.528} C_VEL
LIN {X 0,Y 452.512,Z 521.317,A -85,B 0,C 180,E1 -8178.086,E2 -8178.086} C_VEL
LIN {X 0,Y 452.446,Z 522.094,A -85,B 0,C 180,E1 -8179.257,E2 -8179.257} C_VEL
LIN {X 0,Y 452.416,Z 521.896,A -85,B 0,C 180,E1 -8181.063,E2 -8181.063} C_VEL
LIN {X 0,Y 452.456,Z 521.212,A -85,B 0,C 180,E1 -8181.964,E2 -8181.964} C_VEL
LIN {X 0,Y 452.603,Z 518.889,A -85,B 0,C 180,E1 -8183.611,E2 -8183.611} C_VEL
LIN {X 0,Y 452.625,Z 515.527,A -85,B 0,C 180,E1 -8185.101,E2 -8185.101} C_VEL
LIN {X 0,Y 452.817,Z 511.406,A -85,B 0,C 180,E1 -8186.44,E2 -8186.44} C_VEL
LIN {X 0,Y 453.078,Z 505.132,A -85,B 0,C 180,E1 -8187.999,E2 -8187.999} C_VEL
LIN {X 0,Y 453.438,Z 498.307,A -85,B 0,C 180,E1 -8189.333,E2 -8189.333} C_VEL
LIN {X 0,Y 453.916,Z 489.777,A -85,B 0,C 180,E1 -8190.665,E2 -8190.665} C_VEL
LIN {X 0,Y 454.277,Z 481.07,A -85,B 0,C 180,E1 -8191.773,E2 -8191.773} C_VEL
LIN {X 0,Y 454.753,Z 471.514,A -85,B 0,C 180,E1 -8192.768,E2 -8192.768} C_VEL
LIN {X 0,Y 455.428,Z 461.023,A -85,B 0,C 180,E1 -8193.649,E2 -8193.649} C_VEL
LIN {X 0,Y 455.897,Z 449.438,A -85,B 0,C 180,E1 -8194.42,E2 -8194.42} C_VEL
LIN {X 0,Y 456.344,Z 436.145,A -85,B 0,C 180,E1 -8195.08,E2 -8195.08} C_VEL
LIN {X 0,Y 456.563,Z 426.173,A -85,B 0,C 180,E1 -8195.437,E2 -8195.437} C_VEL
LIN {X 0,Y 456.8,Z 413.286,A -85,B 0,C 180,E1 -8195.739,E2 -8195.739} C_VEL
LIN {X 0,Y 457.588,Z 327.534,A -85,B 0,C 180,E1 -8197.085,E2 -8197.085} C_VEL
LIN {X 0,Y 454.454,Z 311.295,A -85,B 0,C 180,E1 -8197.466,E2 -8197.466} C_VEL
LIN {X 0,Y 454.632,Z 300.943,A -85,B 0,C 180,E1 -8199.565,E2 -8199.565} C_VEL
LIN {X 0,Y 453.566,Z 293.987,A -85,B 0,C 180,E1 -8201.054,E2 -8201.054} C_VEL
LIN {X 0,Y 453.499,Z 293.994,A -85,B 0,C 180,E1 -8203.441,E2 -8203.441} C_VEL
LIN {X 0,Y 453.536,Z 293.992,A -85,B 0,C 180,E1 -8206.196,E2 -8206.196} C_VEL
LIN {X 0,Y 453.515,Z 293.989,A -85,B 0,C 180,E1 -8209.038,E2 -8209.038} C_VEL
LIN {X 0,Y 453.474,Z 293.994,A -85,B 0,C 180,E1 -8211.835,E2 -8211.835} C_VEL
LIN {X 0,Y 453.464,Z 294.001,A -85,B 0,C 180,E1 -8214.736,E2 -8214.736} C_VEL
LIN {X 0,Y 453.459,Z 293.996,A -85,B 0,C 180,E1 -8217.942,E2 -8217.942} C_VEL
LIN {X 0,Y 453.461,Z 294.003,A -85,B 0,C 180,E1 -8220.76,E2 -8220.76} C_VEL
LIN {X 0,Y 453.464,Z 293.994,A -85,B 0,C 180,E1 -8223.913,E2 -8223.913} C_VEL
LIN {X 0,Y 453.447,Z 294.001,A -85,B 0,C 180,E1 -8227.189,E2 -8227.189} C_VEL
LIN {X 0,Y 453.465,Z 293.998,A -85,B 0,C 180,E1 -8230.611,E2 -8230.611} C_VEL
LIN {X 0,Y 453.453,Z 293.996,A -85,B 0,C 180,E1 -8234.221,E2 -8234.221} C_VEL
LIN {X 0,Y 453.442,Z 294.003,A -85,B 0,C 180,E1 -8237.003,E2 -8237.003} C_VEL
LIN {X 0,Y 453.487,Z 293.998,A -85,B 0,C 180,E1 -8239.409,E2 -8239.409} C_VEL
LIN {X 0,Y 453.444,Z 293.999,A -85,B 0,C 180,E1 -8242.81,E2 -8242.81} C_VEL
LIN {X 0,Y 453.469,Z 293.995,A -85,B 0,C 180,E1 -8246.087,E2 -8246.087} C_VEL
LIN {X 0,Y 453.468,Z 293.999,A -85,B 0,C 180,E1 -8249.24,E2 -8249.24} C_VEL
LIN {X 0,Y 453.524,Z 293.988,A -85,B 0,C 180,E1 -8252.297,E2 -8252.297} C_VEL
LIN {X 0,Y 453.491,Z 293.994,A -85,B 0,C 180,E1 -8255.264,E2 -8255.264} C_VEL
LIN {X 0,Y 453.472,Z 293.994,A -85,B 0,C 180,E1 -8258.415,E2 -8258.415} C_VEL
LIN {X 0,Y 453.513,Z 293.988,A -85,B 0,C 180,E1 -8261.008,E2 -8261.008} C_VEL
LIN {X 0,Y 453.568,Z 293.99,A -85,B 0,C 180,E1 -8263.876,E2 -8263.876} C_VEL
LIN {X 0,Y 453.555,Z 293.985,A -85,B 0,C 180,E1 -8267.471,E2 -8267.471} C_VEL
LIN {X 0,Y 453.583,Z 293.979,A -85,B 0,C 180,E1 -8271.087,E2 -8271.087} C_VEL
LIN {X 0,Y 453.642,Z 293.976,A -85,B 0,C 180,E1 -8273.774,E2 -8273.774} C_VEL
LIN {X 0,Y 453.736,Z 293.96,A -85,B 0,C 180,E1 -8277.337,E2 -8277.337} C_VEL
LIN {X 0,Y 453.812,Z 293.955,A -85,B 0,C 180,E1 -8280,E2 -8280} C_VEL
LIN {X 0,Y 453.735,Z 293.965,A -85,B 0,C 180,E1 -8282.663,E2 -8282.663} C_VEL
LIN {X 0,Y 453.668,Z 293.974,A -85,B 0,C 180,E1 -8286.226,E2 -8286.226} C_VEL
LIN {X 0,Y 453.585,Z 293.983,A -85,B 0,C 180,E1 -8288.914,E2 -8288.914} C_VEL
LIN {X 0,Y 453.555,Z 293.99,A -85,B 0,C 180,E1 -8292.529,E2 -8292.529} C_VEL
LIN {X 0,Y 453.537,Z 293.987,A -85,B 0,C 180,E1 -8296.196,E2 -8296.196} C_VEL
LIN {X 0,Y 453.512,Z 293.994,A -85,B 0,C 180,E1 -8299.041,E2 -8299.041} C_VEL
LIN {X 0,Y 453.469,Z 293.994,A -85,B 0,C 180,E1 -8301.837,E2 -8301.837} C_VEL
LIN {X 0,Y 453.507,Z 293.994,A -85,B 0,C 180,E1 -8304.735,E2 -8304.735} C_VEL
LIN {X 0,Y 453.532,Z 293.986,A -85,B 0,C 180,E1 -8307.962,E2 -8307.962} C_VEL
LIN {X 0,Y 453.478,Z 293.996,A -85,B 0,C 180,E1 -8310.76,E2 -8310.76} C_VEL
LIN {X 0,Y 453.471,Z 293.994,A -85,B 0,C 180,E1 -8313.913,E2 -8313.913} C_VEL
LIN {X 0,Y 453.465,Z 294.001,A -85,B 0,C 180,E1 -8317.189,E2 -8317.189} C_VEL
LIN {X 0,Y 453.512,Z 293.996,A -85,B 0,C 180,E1 -8319.448,E2 -8319.448} C_VEL
LIN {X 0,Y 453.464,Z 293.997,A -85,B 0,C 180,E1 -8322.995,E2 -8322.995} C_VEL
LIN {X 0,Y 453.462,Z 294,A -85,B 0,C 180,E1 -8325.78,E2 -8325.78} C_VEL
LIN {X 0,Y 453.475,Z 293.994,A -85,B 0,C 180,E1 -8328.21,E2 -8328.21} C_VEL
LIN {X 0,Y 453.484,Z 293.992,A -85,B 0,C 180,E1 -8330.795,E2 -8330.795} C_VEL
LIN {X 0,Y 453.452,Z 294.002,A -85,B 0,C 180,E1 -8333.918,E2 -8333.918} C_VEL
LIN {X 0,Y 453.481,Z 293.993,A -85,B 0,C 180,E1 -8337.152,E2 -8337.152} C_VEL
LIN {X 0,Y 453.474,Z 293.999,A -85,B 0,C 180,E1 -8340.269,E2 -8340.269} C_VEL
LIN {X 0,Y 453.538,Z 293.99,A -85,B 0,C 180,E1 -8343.297,E2 -8343.297} C_VEL
LIN {X 0,Y 453.6,Z 294.194,A -85,B 0,C 180,E1 -8343.742,E2 -8343.742} C_VEL
LIN {X 0,Y 455.766,Z 305.615,A -85,B 0,C 180,E1 -8345.933,E2 -8345.933} C_VEL
LIN {X 0,Y 455.423,Z 315.246,A -85,B 0,C 180,E1 -8347.655,E2 -8347.655} C_VEL
LIN {X 0,Y 454.739,Z 331.442,A -85,B 0,C 180,E1 -8350.52,E2 -8350.52} C_VEL
LIN {X 0,Y 454.222,Z 342.961,A -85,B 0,C 180,E1 -8352.539,E2 -8352.539} C_VEL
LIN {X 0,Y 457.334,Z 364.043,A -85,B 0,C 180,E1 -8353.001,E2 -8353.001} C_VEL
LIN {X 0,Y 456.6,Z 451.899,A -85,B 0,C 180,E1 -8354.403,E2 -8354.403} C_VEL
LIN {X 0,Y 456.258,Z 465.079,A -85,B 0,C 180,E1 -8354.792,E2 -8354.792} C_VEL
LIN {X 0,Y 455.786,Z 477.208,A -85,B 0,C 180,E1 -8355.318,E2 -8355.318} C_VEL
LIN {X 0,Y 455.227,Z 489.45,A -85,B 0,C 180,E1 -8356.042,E2 -8356.042} C_VEL
LIN {X 0,Y 454.672,Z 501.098,A -85,B 0,C 180,E1 -8356.939,E2 -8356.939} C_VEL
LIN {X 0,Y 454.179,Z 511.518,A -85,B 0,C 180,E1 -8357.943,E2 -8357.943} C_VEL
LIN {X 0,Y 453.658,Z 520.9,A -85,B 0,C 180,E1 -8359.061,E2 -8359.061} C_VEL
LIN {X 0,Y 453.188,Z 529.98,A -85,B 0,C 180,E1 -8360.404,E2 -8360.404} C_VEL
LIN {X 0,Y 452.869,Z 537.294,A -85,B 0,C 180,E1 -8361.747,E2 -8361.747} C_VEL
LIN {X 0,Y 452.69,Z 542.236,A -85,B 0,C 180,E1 -8362.866,E2 -8362.866} C_VEL
LIN {X 0,Y 452.554,Z 547.035,A -85,B 0,C 180,E1 -8364.207,E2 -8364.207} C_VEL
LIN {X 0,Y 452.486,Z 550.707,A -85,B 0,C 180,E1 -8365.546,E2 -8365.546} C_VEL
LIN {X 0,Y 452.484,Z 552.604,A -85,B 0,C 180,E1 -8366.439,E2 -8366.439} C_VEL
LIN {X 0,Y 452.508,Z 554.04,A -85,B 0,C 180,E1 -8367.33,E2 -8367.33} C_VEL
LIN {X 0,Y 452.457,Z 555.681,A -85,B 0,C 180,E1 -8369.11,E2 -8369.11} C_VEL
LIN {X 0,Y 452.465,Z 555.92,A -85,B 0,C 180,E1 -8370,E2 -8370} C_VEL
LIN {X 0,Y 452.43,Z 555.731,A -85,B 0,C 180,E1 -8370.891,E2 -8370.891} C_VEL
LIN {X 0,Y 452.508,Z 554.158,A -85,B 0,C 180,E1 -8372.671,E2 -8372.671} C_VEL
LIN {X 0,Y 452.482,Z 552.78,A -85,B 0,C 180,E1 -8373.562,E2 -8373.562} C_VEL
LIN {X 0,Y 452.545,Z 549.873,A -85,B 0,C 180,E1 -8374.9,E2 -8374.9} C_VEL
LIN {X 0,Y 452.611,Z 545.424,A -85,B 0,C 180,E1 -8376.396,E2 -8376.396} C_VEL
LIN {X 0,Y 452.779,Z 540.877,A -85,B 0,C 180,E1 -8377.582,E2 -8377.582} C_VEL
LIN {X 0,Y 453.054,Z 534.527,A -85,B 0,C 180,E1 -8378.924,E2 -8378.924} C_VEL
LIN {X 0,Y 453.42,Z 526.592,A -85,B 0,C 180,E1 -8380.268,E2 -8380.268} C_VEL
LIN {X 0,Y 453.95,Z 518.528,A -85,B 0,C 180,E1 -8381.385,E2 -8381.385} C_VEL
LIN {X 0,Y 454.497,Z 508.705,A -85,B 0,C 180,E1 -8382.503,E2 -8382.503} C_VEL
LIN {X 0,Y 455.069,Z 497.749,A -85,B 0,C 180,E1 -8383.509,E2 -8383.509} C_VEL
LIN {X 0,Y 455.715,Z 485.266,A -85,B 0,C 180,E1 -8384.4,E2 -8384.4} C_VEL
LIN {X 0,Y 456.346,Z 473.003,A -85,B 0,C 180,E1 -8385.064,E2 -8385.064} C_VEL
LIN {X 0,Y 456.816,Z 460.063,A -85,B 0,C 180,E1 -8385.562,E2 -8385.562} C_VEL
LIN {X 0,Y 457.124,Z 446.297,A -85,B 0,C 180,E1 -8385.894,E2 -8385.894} C_VEL
LIN {X 0,Y 457.848,Z 364.68,A -85,B 0,C 180,E1 -8387.193,E2 -8387.193} C_VEL
LIN {X 0,Y 454.699,Z 344.39,A -85,B 0,C 180,E1 -8387.661,E2 -8387.661} C_VEL
LIN {X 0,Y 454.443,Z 342.809,A -85,B 0,C 180,E1 -8387.703,E2 -8387.703} C_VEL
LIN {X 0,Y 455.293,Z 325.423,A -85,B 0,C 180,E1 -8390.796,E2 -8390.796} C_VEL
LIN {X 0,Y 456.193,Z 308.523,A -85,B 0,C 180,E1 -8393.849,E2 -8393.849} C_VEL
LIN {X 0,Y 455.211,Z 301.979,A -85,B 0,C 180,E1 -8395.124,E2 -8395.124} C_VEL
LIN {X 0,Y 453.564,Z 293.991,A -85,B 0,C 180,E1 -8396.765,E2 -8396.765} C_VEL
LIN {X 0,Y 453.475,Z 294.005,A -85,B 0,C 180,E1 -8399.785,E2 -8399.785} C_VEL
LIN {X 0,Y 453.492,Z 293.992,A -85,B 0,C 180,E1 -8403.189,E2 -8403.189} C_VEL
LIN {X 0,Y 453.455,Z 294.004,A -85,B 0,C 180,E1 -8406.299,E2 -8406.299} C_VEL
LIN {X 0,Y 453.484,Z 293.994,A -85,B 0,C 180,E1 -8409.45,E2 -8409.45} C_VEL
LIN {X 0,Y 453.477,Z 293.996,A -85,B 0,C 180,E1 -8411.935,E2 -8411.935} C_VEL
LIN {X 0,Y 453.485,Z 293.994,A -85,B 0,C 180,E1 -8415.471,E2 -8415.471} C_VEL
LIN {X 0,Y 453.479,Z 293.995,A -85,B 0,C 180,E1 -8418.209,E2 -8418.209} C_VEL
LIN {X 0,Y 453.491,Z 293.998,A -85,B 0,C 180,E1 -8420.794,E2 -8420.794} C_VEL
LIN {X 0,Y 453.454,Z 293.996,A -85,B 0,C 180,E1 -8423.917,E2 -8423.917} C_VEL
LIN {X 0,Y 453.482,Z 293.999,A -85,B 0,C 180,E1 -8427.151,E2 -8427.151} C_VEL
LIN {X 0,Y 453.474,Z 293.992,A -85,B 0,C 180,E1 -8430.268,E2 -8430.268} C_VEL
LIN {X 0,Y 453.504,Z 293.994,A -85,B 0,C 180,E1 -8433.294,E2 -8433.294} C_VEL
LIN {X 0,Y 453.501,Z 293.99,A -85,B 0,C 180,E1 -8436.239,E2 -8436.239} C_VEL
LIN {X 0,Y 453.482,Z 293.997,A -85,B 0,C 180,E1 -8439.117,E2 -8439.117} C_VEL
LIN {X 0,Y 453.51,Z 293.99,A -85,B 0,C 180,E1 -8441.944,E2 -8441.944} C_VEL
LIN {X 0,Y 453.54,Z 293.984,A -85,B 0,C 180,E1 -8444.726,E2 -8444.726} C_VEL
LIN {X 0,Y 453.558,Z 293.982,A -85,B 0,C 180,E1 -8448.379,E2 -8448.379} C_VEL
LIN {X 0,Y 453.651,Z 293.975,A -85,B 0,C 180,E1 -8451.985,E2 -8451.985} C_VEL
LIN {X 0,Y 453.668,Z 293.964,A -85,B 0,C 180,E1 -8454.667,E2 -8454.667} C_VEL
LIN {X 0,Y 453.743,Z 293.959,A -85,B 0,C 180,E1 -8457.337,E2 -8457.337} C_VEL
LIN {X 0,Y 453.821,Z 293.952,A -85,B 0,C 180,E1 -8460,E2 -8460} C_VEL
LIN {X 0,Y 453.742,Z 293.956,A -85,B 0,C 180,E1 -8462.663,E2 -8462.663} C_VEL
LIN {X 0,Y 453.667,Z 293.974,A -85,B 0,C 180,E1 -8466.225,E2 -8466.225} C_VEL
LIN {X 0,Y 453.59,Z 293.979,A -85,B 0,C 180,E1 -8468.913,E2 -8468.913} C_VEL
LIN {X 0,Y 453.562,Z 293.986,A -85,B 0,C 180,E1 -8472.529,E2 -8472.529} C_VEL
LIN {X 0,Y 453.543,Z 293.988,A -85,B 0,C 180,E1 -8476.196,E2 -8476.196} C_VEL
LIN {X 0,Y 453.518,Z 293.991,A -85,B 0,C 180,E1 -8479.041,E2 -8479.041} C_VEL
LIN {X 0,Y 453.475,Z 293.993,A -85,B 0,C 180,E1 -8481.836,E2 -8481.836} C_VEL
LIN {X 0,Y 453.513,Z 293.992,A -85,B 0,C 180,E1 -8484.734,E2 -8484.734} C_VEL
LIN {X 0,Y 453.531,Z 293.983,A -85,B 0,C 180,E1 -8487.96,E2 -8487.96} C_VEL
LIN {X 0,Y 453.464,Z 293.994,A -85,B 0,C 180,E1 -8491.525,E2 -8491.525} C_VEL
LIN {X 0,Y 453.486,Z 293.995,A -85,B 0,C 180,E1 -8494.777,E2 -8494.777} C_VEL
LIN {X 0,Y 453.462,Z 293.995,A -85,B 0,C 180,E1 -8498.312,E2 -8498.312} C_VEL
LIN {X 0,Y 453.493,Z 293.99,A -85,B 0,C 180,E1 -8500.609,E2 -8500.609} C_VEL
LIN {X 0,Y 453.454,Z 294.002,A -85,B 0,C 180,E1 -8503.244,E2 -8503.244} C_VEL
LIN {X 0,Y 453.461,Z 294,A -85,B 0,C 180,E1 -8505.779,E2 -8505.779} C_VEL
LIN {X 0,Y 453.479,Z 293.994,A -85,B 0,C 180,E1 -8508.209,E2 -8508.209} C_VEL
LIN {X 0,Y 453.487,Z 293.995,A -85,B 0,C 180,E1 -8510.795,E2 -8510.795} C_VEL
LIN {X 0,Y 453.454,Z 294.001,A -85,B 0,C 180,E1 -8513.917,E2 -8513.917} C_VEL
LIN {X 0,Y 453.484,Z 293.998,A -85,B 0,C 180,E1 -8517.151,E2 -8517.151} C_VEL
LIN {X 0,Y 453.516,Z 294.144,A -85,B 0,C 180,E1 -8518.782,E2 -8518.782} C_VEL
LIN {X 0,Y 454.904,Z 301.506,A -85,B 0,C 180,E1 -8520.371,E2 -8520.371} C_VEL
LIN {X 0,Y 454.684,Z 311.398,A -85,B 0,C 180,E1 -8522.356,E2 -8522.356} C_VEL
LIN {X 0,Y 458.125,Z 327.942,A -85,B 0,C 180,E1 -8522.783,E2 -8522.783} C_VEL
LIN {X 0,Y 457.193,Z 418.249,A -85,B 0,C 180,E1 -8524.231,E2 -8524.231} C_VEL
LIN {X 0,Y 456.83,Z 431.271,A -85,B 0,C 180,E1 -8524.606,E2 -8524.606} C_VEL
LIN {X 0,Y 456.525,Z 443.811,A -85,B 0,C 180,E1 -8525.155,E2 -8525.155} C_VEL
LIN {X 0,Y 456.093,Z 454.379,A -85,B 0,C 180,E1 -8525.769,E2 -8525.769} C_VEL
LIN {X 0,Y 455.226,Z 459.607,A -85,B 0,C 180,E1 -8526.1,E2 -8526.1} C_VEL
LIN {X 0,Y 451.977,Z 467.901,A -85,B 0,C 180,E1 -8526.656,E2 -8526.656} C_VEL
LIN {X 0,Y 448.712,Z 475.73,A -85,B 0,C 180,E1 -8527.306,E2 -8527.306} C_VEL
LIN {X 0,Y 447.823,Z 480.221,A -85,B 0,C 180,E1 -8527.78,E2 -8527.78} C_VEL
LIN {X 0,Y 447.18,Z 490.126,A -85,B 0,C 180,E1 -8529.05,E2 -8529.05} C_VEL
LIN {X 0,Y 446.752,Z 497.603,A -85,B 0,C 180,E1 -8530.231,E2 -8530.231} C_VEL
LIN {X 0,Y 446.243,Z 504.871,A -85,B 0,C 180,E1 -8531.64,E2 -8531.64} C_VEL
LIN {X 0,Y 445.906,Z 510.602,A -85,B 0,C 180,E1 -8533.047,E2 -8533.047} C_VEL
LIN {X 0,Y 445.689,Z 515.067,A -85,B 0,C 180,E1 -8534.45,E2 -8534.45} C_VEL
LIN {X 0,Y 445.585,Z 517.41,A -85,B 0,C 180,E1 -8535.382,E2 -8535.382} C_VEL
LIN {X 0,Y 445.447,Z 519.304,A -85,B 0,C 180,E1 -8536.31,E2 -8536.31} C_VEL
LIN {X 0,Y 445.428,Z 521.58,A -85,B 0,C 180,E1 -8538.026,E2 -8538.026} C_VEL
LIN {X 0,Y 445.356,Z 522.295,A -85,B 0,C 180,E1 -8539.084,E2 -8539.084} C_VEL
LIN {X 0,Y 445.309,Z 522.482,A -85,B 0,C 180,E1 -8540.002,E2 -8540.002} C_VEL
LIN {X 0,Y 445.351,Z 521.596,A -85,B 0,C 180,E1 -8541.834,E2 -8541.834} C_VEL
LIN {X 0,Y 445.442,Z 520.569,A -85,B 0,C 180,E1 -8542.748,E2 -8542.748} C_VEL
LIN {X 0,Y 445.529,Z 519.118,A -85,B 0,C 180,E1 -8543.66,E2 -8543.66} C_VEL
LIN {X 0,Y 445.553,Z 516.151,A -85,B 0,C 180,E1 -8545.023,E2 -8545.023} C_VEL
LIN {X 0,Y 445.74,Z 512.136,A -85,B 0,C 180,E1 -8546.384,E2 -8546.384} C_VEL
LIN {X 0,Y 446.006,Z 505.977,A -85,B 0,C 180,E1 -8547.968,E2 -8547.968} C_VEL
LIN {X 0,Y 446.351,Z 499.282,A -85,B 0,C 180,E1 -8549.323,E2 -8549.323} C_VEL
LIN {X 0,Y 446.852,Z 490.972,A -85,B 0,C 180,E1 -8550.675,E2 -8550.675} C_VEL
LIN {X 0,Y 447.226,Z 482.448,A -85,B 0,C 180,E1 -8551.801,E2 -8551.801} C_VEL
LIN {X 0,Y 447.775,Z 471.952,A -85,B 0,C 180,E1 -8552.923,E2 -8552.923} C_VEL
LIN {X 0,Y 448.49,Z 461.491,A -85,B 0,C 180,E1 -8553.818,E2 -8553.818} C_VEL
LIN {X 0,Y 448.982,Z 449.981,A -85,B 0,C 180,E1 -8554.601,E2 -8554.601} C_VEL
LIN {X 0,Y 449.416,Z 438.047,A -85,B 0,C 180,E1 -8555.215,E2 -8555.215} C_VEL
LIN {X 0,Y 449.619,Z 426.974,A -85,B 0,C 180,E1 -8555.634,E2 -8555.634} C_VEL
LIN {X 0,Y 449.921,Z 414.371,A -85,B 0,C 180,E1 -8555.939,E2 -8555.939} C_VEL
LIN {X 0,Y 450.65,Z 327.848,A -85,B 0,C 180,E1 -8557.323,E2 -8557.323} C_VEL
LIN {X 0,Y 447.499,Z 311.476,A -85,B 0,C 180,E1 -8557.724,E2 -8557.724} C_VEL
LIN {X 0,Y 447.645,Z 301.774,A -85,B 0,C 180,E1 -8559.716,E2 -8559.716} C_VEL
LIN {X 0,Y 446.496,Z 294.868,A -85,B 0,C 180,E1 -8561.232,E2 -8561.232} C_VEL
LIN {X 0,Y 446.459,Z 294.872,A -85,B 0,C 180,E1 -8563.657,E2 -8563.657} C_VEL
LIN {X 0,Y 446.483,Z 294.871,A -85,B 0,C 180,E1 -8566.459,E2 -8566.459} C_VEL
LIN {X 0,Y 446.466,Z 294.866,A -85,B 0,C 180,E1 -8569.303,E2 -8569.303} C_VEL
LIN {X 0,Y 446.415,Z 294.877,A -85,B 0,C 180,E1 -8572.199,E2 -8572.199} C_VEL
LIN {X 0,Y 446.416,Z 294.874,A -85,B 0,C 180,E1 -8575.154,E2 -8575.154} C_VEL
LIN {X 0,Y 446.433,Z 294.873,A -85,B 0,C 180,E1 -8578.181,E2 -8578.181} C_VEL
LIN {X 0,Y 446.408,Z 294.875,A -85,B 0,C 180,E1 -8581.3,E2 -8581.3} C_VEL
LIN {X 0,Y 446.419,Z 294.876,A -85,B 0,C 180,E1 -8584.523,E2 -8584.523} C_VEL
LIN {X 0,Y 446.407,Z 294.874,A -85,B 0,C 180,E1 -8588.078,E2 -8588.078} C_VEL
LIN {X 0,Y 446.4,Z 294.878,A -85,B 0,C 180,E1 -8591.393,E2 -8591.393} C_VEL
LIN {X 0,Y 446.444,Z 294.878,A -85,B 0,C 180,E1 -8595.103,E2 -8595.103} C_VEL
LIN {X 0,Y 446.412,Z 294.874,A -85,B 0,C 180,E1 -8598.607,E2 -8598.607} C_VEL
LIN {X 0,Y 446.405,Z 294.875,A -85,B 0,C 180,E1 -8601.921,E2 -8601.921} C_VEL
LIN {X 0,Y 446.422,Z 294.879,A -85,B 0,C 180,E1 -8605.476,E2 -8605.476} C_VEL
LIN {X 0,Y 446.408,Z 294.874,A -85,B 0,C 180,E1 -8608.699,E2 -8608.699} C_VEL
LIN {X 0,Y 446.477,Z 294.87,A -85,B 0,C 180,E1 -8611.821,E2 -8611.821} C_VEL
LIN {X 0,Y 446.434,Z 294.87,A -85,B 0,C 180,E1 -8614.846,E2 -8614.846} C_VEL
LIN {X 0,Y 446.44,Z 294.871,A -85,B 0,C 180,E1 -8618.245,E2 -8618.245} C_VEL
LIN {X 0,Y 446.449,Z 294.874,A -85,B 0,C 180,E1 -8621.649,E2 -8621.649} C_VEL
LIN {X 0,Y 446.507,Z 294.862,A -85,B 0,C 180,E1 -8624.48,E2 -8624.48} C_VEL
LIN {X 0,Y 446.509,Z 294.867,A -85,B 0,C 180,E1 -8628.193,E2 -8628.193} C_VEL
LIN {X 0,Y 446.529,Z 294.858,A -85,B 0,C 180,E1 -8630.945,E2 -8630.945} C_VEL
LIN {X 0,Y 446.61,Z 294.851,A -85,B 0,C 180,E1 -8633.676,E2 -8633.676} C_VEL
LIN {X 0,Y 446.683,Z 294.839,A -85,B 0,C 180,E1 -8637.295,E2 -8637.295} C_VEL
LIN {X 0,Y 446.782,Z 294.831,A -85,B 0,C 180,E1 -8640,E2 -8640} C_VEL
LIN {X 0,Y 446.682,Z 294.843,A -85,B 0,C 180,E1 -8642.706,E2 -8642.706} C_VEL
LIN {X 0,Y 446.638,Z 294.851,A -85,B 0,C 180,E1 -8646.324,E2 -8646.324} C_VEL
LIN {X 0,Y 446.531,Z 294.86,A -85,B 0,C 180,E1 -8649.056,E2 -8649.056} C_VEL
LIN {X 0,Y 446.513,Z 294.868,A -85,B 0,C 180,E1 -8652.73,E2 -8652.73} C_VEL
LIN {X 0,Y 446.488,Z 294.865,A -85,B 0,C 180,E1 -8656.228,E2 -8656.228} C_VEL
LIN {X 0,Y 446.461,Z 294.869,A -85,B 0,C 180,E1 -8659.304,E2 -8659.304} C_VEL
LIN {X 0,Y 446.41,Z 294.874,A -85,B 0,C 180,E1 -8662.2,E2 -8662.2} C_VEL
LIN {X 0,Y 446.452,Z 294.874,A -85,B 0,C 180,E1 -8665.153,E2 -8665.153} C_VEL
LIN {X 0,Y 446.478,Z 294.865,A -85,B 0,C 180,E1 -8668.179,E2 -8668.179} C_VEL
LIN {X 0,Y 446.428,Z 294.877,A -85,B 0,C 180,E1 -8671.3,E2 -8671.3} C_VEL
LIN {X 0,Y 446.424,Z 294.872,A -85,B 0,C 180,E1 -8674.524,E2 -8674.524} C_VEL
LIN {X 0,Y 446.425,Z 294.872,A -85,B 0,C 180,E1 -8678.083,E2 -8678.083} C_VEL
LIN {X 0,Y 446.423,Z 294.874,A -85,B 0,C 180,E1 -8680.919,E2 -8680.919} C_VEL
LIN {X 0,Y 446.419,Z 294.876,A -85,B 0,C 180,E1 -8683.844,E2 -8683.844} C_VEL
LIN {X 0,Y 446.395,Z 294.875,A -85,B 0,C 180,E1 -8686.404,E2 -8686.404} C_VEL
LIN {X 0,Y 446.423,Z 294.873,A -85,B 0,C 180,E1 -8689.083,E2 -8689.083} C_VEL
LIN {X 0,Y 446.404,Z 294.877,A -85,B 0,C 180,E1 -8692.122,E2 -8692.122} C_VEL
LIN {X 0,Y 446.427,Z 294.875,A -85,B 0,C 180,E1 -8695.478,E2 -8695.478} C_VEL
LIN {X 0,Y 446.414,Z 294.873,A -85,B 0,C 180,E1 -8698.701,E2 -8698.701} C_VEL
LIN {X 0,Y 446.484,Z 294.871,A -85,B 0,C 180,E1 -8701.822,E2 -8701.822} C_VEL
LIN {X 0,Y 446.527,Z 294.901,A -85,B 0,C 180,E1 -8703.523,E2 -8703.523} C_VEL
LIN {X 0,Y 448.864,Z 307.535,A -85,B 0,C 180,E1 -8705.979,E2 -8705.979} C_VEL
LIN {X 0,Y 448.102,Z 324.791,A -85,B 0,C 180,E1 -8709.096,E2 -8709.096} C_VEL
LIN {X 0,Y 447.267,Z 342.667,A -85,B 0,C 180,E1 -8712.285,E2 -8712.285} C_VEL
LIN {X 0,Y 450.494,Z 365.199,A -85,B 0,C 180,E1 -8712.788,E2 -8712.788} C_VEL
LIN {X 0,Y 449.715,Z 451.646,A -85,B 0,C 180,E1 -8714.187,E2 -8714.187} C_VEL
LIN {X 0,Y 449.363,Z 464.829,A -85,B 0,C 180,E1 -8714.582,E2 -8714.582} C_VEL
LIN {X 0,Y 448.846,Z 477.526,A -85,B 0,C 180,E1 -8715.144,E2 -8715.144} C_VEL
LIN {X 0,Y 448.294,Z 488.802,A -85,B 0,C 180,E1 -8715.821,E2 -8715.821} C_VEL
LIN {X 0,Y 447.713,Z 500.371,A -85,B 0,C 180,E1 -8716.718,E2 -8716.718} C_VEL
LIN {X 0,Y 447.139,Z 510.998,A -85,B 0,C 180,E1 -8717.75,E2 -8717.75} C_VEL
LIN {X 0,Y 446.662,Z 520.449,A -85,B 0,C 180,E1 -8718.887,E2 -8718.887} C_VEL
LIN {X 0,Y 446.147,Z 529.563,A -85,B 0,C 180,E1 -8720.251,E2 -8720.251} C_VEL
LIN {X 0,Y 445.823,Z 536.907,A -85,B 0,C 180,E1 -8721.616,E2 -8721.616} C_VEL
LIN {X 0,Y 445.613,Z 541.874,A -85,B 0,C 180,E1 -8722.752,E2 -8722.752} C_VEL
LIN {X 0,Y 445.457,Z 546.241,A -85,B 0,C 180,E1 -8723.971,E2 -8723.971} C_VEL
LIN {X 0,Y 445.412,Z 550.388,A -85,B 0,C 180,E1 -8725.476,E2 -8725.476} C_VEL
LIN {X 0,Y 445.384,Z 552.294,A -85,B 0,C 180,E1 -8726.382,E2 -8726.382} C_VEL
LIN {X 0,Y 445.433,Z 553.747,A -85,B 0,C 180,E1 -8727.287,E2 -8727.287} C_VEL
LIN {X 0,Y 445.366,Z 555.404,A -85,B 0,C 180,E1 -8729.096,E2 -8729.096} C_VEL
LIN {X 0,Y 445.371,Z 555.651,A -85,B 0,C 180,E1 -8730,E2 -8730} C_VEL
LIN {X 0,Y 445.341,Z 555.478,A -85,B 0,C 180,E1 -8730.905,E2 -8730.905} C_VEL
LIN {X 0,Y 445.433,Z 553.922,A -85,B 0,C 180,E1 -8732.713,E2 -8732.713} C_VEL
LIN {X 0,Y 445.38,Z 552.551,A -85,B 0,C 180,E1 -8733.619,E2 -8733.619} C_VEL
LIN {X 0,Y 445.474,Z 549.663,A -85,B 0,C 180,E1 -8734.978,E2 -8734.978} C_VEL
LIN {X 0,Y 445.53,Z 545.602,A -85,B 0,C 180,E1 -8736.386,E2 -8736.386} C_VEL
LIN {X 0,Y 445.715,Z 540.709,A -85,B 0,C 180,E1 -8737.703,E2 -8737.703} C_VEL
LIN {X 0,Y 445.989,Z 534.391,A -85,B 0,C 180,E1 -8739.067,E2 -8739.067} C_VEL
LIN {X 0,Y 446.409,Z 526.496,A -85,B 0,C 180,E1 -8740.431,E2 -8740.431} C_VEL
LIN {X 0,Y 447.087,Z 516.687,A -85,B 0,C 180,E1 -8741.792,E2 -8741.792} C_VEL
LIN {X 0,Y 447.677,Z 507.49,A -85,B 0,C 180,E1 -8742.826,E2 -8742.826} C_VEL
LIN {X 0,Y 448.157,Z 497.826,A -85,B 0,C 180,E1 -8743.721,E2 -8743.721} C_VEL
LIN {X 0,Y 448.843,Z 485.442,A -85,B 0,C 180,E1 -8744.625,E2 -8744.625} C_VEL
LIN {X 0,Y 449.5,Z 473.313,A -85,B 0,C 180,E1 -8745.299,E2 -8745.299} C_VEL
LIN {X 0,Y 450.013,Z 460.729,A -85,B 0,C 180,E1 -8745.803,E2 -8745.803} C_VEL
LIN {X 0,Y 450.35,Z 447.573,A -85,B 0,C 180,E1 -8746.14,E2 -8746.14} C_VEL
LIN {X 0,Y 451.126,Z 365.232,A -85,B 0,C 180,E1 -8747.475,E2 -8747.475} C_VEL
LIN {X 0,Y 447.792,Z 344.24,A -85,B 0,C 180,E1 -8747.975,E2 -8747.975} C_VEL
LIN {X 0,Y 447.507,Z 342.423,A -85,B 0,C 180,E1 -8748.04,E2 -8748.04} C_VEL
LIN {X 0,Y 448.495,Z 324.047,A -85,B 0,C 180,E1 -8751.367,E2 -8751.367} C_VEL
LIN {X 0,Y 449.28,Z 309.737,A -85,B 0,C 180,E1 -8753.999,E2 -8753.999} C_VEL
LIN {X 0,Y 448.01,Z 301.923,A -85,B 0,C 180,E1 -8755.556,E2 -8755.556} C_VEL
LIN {X 0,Y 446.516,Z 294.869,A -85,B 0,C 180,E1 -8757.046,E2 -8757.046} C_VEL
LIN {X 0,Y 446.43,Z 294.878,A -85,B 0,C 180,E1 -8760.25,E2 -8760.25} C_VEL
LIN {X 0,Y 446.447,Z 294.87,A -85,B 0,C 180,E1 -8763.454,E2 -8763.454} C_VEL
LIN {X 0,Y 446.403,Z 294.88,A -85,B 0,C 180,E1 -8766.745,E2 -8766.745} C_VEL
LIN {X 0,Y 446.443,Z 294.876,A -85,B 0,C 180,E1 -8770.198,E2 -8770.198} C_VEL
LIN {X 0,Y 446.43,Z 294.878,A -85,B 0,C 180,E1 -8772.604,E2 -8772.604} C_VEL
LIN {X 0,Y 446.452,Z 294.872,A -85,B 0,C 180,E1 -8775.104,E2 -8775.104} C_VEL
LIN {X 0,Y 446.428,Z 294.878,A -85,B 0,C 180,E1 -8778.609,E2 -8778.609} C_VEL
LIN {X 0,Y 446.442,Z 294.876,A -85,B 0,C 180,E1 -8780.972,E2 -8780.972} C_VEL
LIN {X 0,Y 446.419,Z 294.874,A -85,B 0,C 180,E1 -8784.374,E2 -8784.374} C_VEL
LIN {X 0,Y 446.422,Z 294.873,A -85,B 0,C 180,E1 -8787.638,E2 -8787.638} C_VEL
LIN {X 0,Y 446.448,Z 294.871,A -85,B 0,C 180,E1 -8790.79,E2 -8790.79} C_VEL
LIN {X 0,Y 446.477,Z 294.866,A -85,B 0,C 180,E1 -8793.848,E2 -8793.848} C_VEL
LIN {X 0,Y 446.428,Z 294.873,A -85,B 0,C 180,E1 -8796.823,E2 -8796.823} C_VEL
LIN {X 0,Y 446.443,Z 294.872,A -85,B 0,C 180,E1 -8799.737,E2 -8799.737} C_VEL
LIN {X 0,Y 446.462,Z 294.866,A -85,B 0,C 180,E1 -8802.597,E2 -8802.597} C_VEL
LIN {X 0,Y 446.471,Z 294.868,A -85,B 0,C 180,E1 -8805.412,E2 -8805.412} C_VEL
LIN {X 0,Y 446.516,Z 294.86,A -85,B 0,C 180,E1 -8808.193,E2 -8808.193} C_VEL
LIN {X 0,Y 446.599,Z 294.855,A -85,B 0,C 180,E1 -8811.858,E2 -8811.858} C_VEL
LIN {X 0,Y 446.643,Z 294.839,A -85,B 0,C 180,E1 -8814.582,E2 -8814.582} C_VEL
LIN {X 0,Y 446.662,Z 294.839,A -85,B 0,C 180,E1 -8818.197,E2 -8818.197} C_VEL
LIN {X 0,Y 446.791,Z 294.827,A -85,B 0,C 180,E1 -8820,E2 -8820} C_VEL
LIN {X 0,Y 446.69,Z 294.834,A -85,B 0,C 180,E1 -8822.705,E2 -8822.705} C_VEL
LIN {X 0,Y 446.637,Z 294.848,A -85,B 0,C 180,E1 -8826.324,E2 -8826.324} C_VEL
LIN {X 0,Y 446.536,Z 294.857,A -85,B 0,C 180,E1 -8829.055,E2 -8829.055} C_VEL
LIN {X 0,Y 446.52,Z 294.863,A -85,B 0,C 180,E1 -8832.73,E2 -8832.73} C_VEL
LIN {X 0,Y 446.495,Z 294.867,A -85,B 0,C 180,E1 -8836.228,E2 -8836.228} C_VEL
LIN {X 0,Y 446.468,Z 294.867,A -85,B 0,C 180,E1 -8839.303,E2 -8839.303} C_VEL
LIN {X 0,Y 446.417,Z 294.874,A -85,B 0,C 180,E1 -8842.2,E2 -8842.2} C_VEL
LIN {X 0,Y 446.457,Z 294.871,A -85,B 0,C 180,E1 -8845.152,E2 -8845.152} C_VEL
LIN {X 0,Y 446.483,Z 294.862,A -85,B 0,C 180,E1 -8848.179,E2 -8848.179} C_VEL
LIN {X 0,Y 446.418,Z 294.87,A -85,B 0,C 180,E1 -8851.775,E2 -8851.775} C_VEL
LIN {X 0,Y 446.427,Z 294.872,A -85,B 0,C 180,E1 -8854.523,E2 -8854.523} C_VEL
LIN {X 0,Y 446.414,Z 294.873,A -85,B 0,C 180,E1 -8858.079,E2 -8858.079} C_VEL
LIN {X 0,Y 446.426,Z 294.873,A -85,B 0,C 180,E1 -8860.918,E2 -8860.918} C_VEL
LIN {X 0,Y 446.399,Z 294.878,A -85,B 0,C 180,E1 -8863.846,E2 -8863.846} C_VEL
LIN {X 0,Y 446.395,Z 294.876,A -85,B 0,C 180,E1 -8866.404,E2 -8866.404} C_VEL
LIN {X 0,Y 446.426,Z 294.875,A -85,B 0,C 180,E1 -8869.083,E2 -8869.083} C_VEL
LIN {X 0,Y 446.407,Z 294.875,A -85,B 0,C 180,E1 -8872.121,E2 -8872.121} C_VEL
LIN {X 0,Y 446.43,Z 294.877,A -85,B 0,C 180,E1 -8875.477,E2 -8875.477} C_VEL
LIN {X 0,Y 446.485,Z 295.016,A -85,B 0,C 180,E1 -8878.53,E2 -8878.53} C_VEL
LIN {X 0,Y 447.891,Z 302.247,A -85,B 0,C 180,E1 -8880.119,E2 -8880.119} C_VEL
LIN {X 0,Y 447.872,Z 309.53,A -85,B 0,C 180,E1 -8881.616,E2 -8881.616} C_VEL
LIN {X 0,Y 447.842,Z 311.758,A -85,B 0,C 180,E1 -8882.043,E2 -8882.043} C_VEL
LIN {X 0,Y 451.432,Z 328.793,A -85,B 0,C 180,E1 -8882.496,E2 -8882.496} C_VEL
LIN {X 0,Y 450.428,Z 419.1,A -85,B 0,C 180,E1 -8883.97,E2 -8883.97} C_VEL
LIN {X 0,Y 450.015,Z 432.686,A -85,B 0,C 180,E1 -8884.38,E2 -8884.38} C_VEL
LIN {X 0,Y 449.672,Z 445.719,A -85,B 0,C 180,E1 -8884.978,E2 -8884.978} C_VEL
LIN {X 0,Y 449.202,Z 456.428,A -85,B 0,C 180,E1 -8885.637,E2 -8885.637} C_VEL
LIN {X 0,Y 448.514,Z 468.27,A -85,B 0,C 180,E1 -8886.571,E2 -8886.571} C_VEL
LIN {X 0,Y 447.873,Z 479.175,A -85,B 0,C 180,E1 -8887.658,E2 -8887.658} C_VEL
LIN {X 0,Y 447.823,Z 480.221,A -85,B 0,C 180,E1 -8887.78,E2 -8887.78} C_VEL
LIN {X 0,Y 446.968,Z 484.598,A -85,B 0,C 180,E1 -8888.285,E2 -8888.285} C_VEL
LIN {X 0,Y 443.779,Z 491.421,A -85,B 0,C 180,E1 -8889.119,E2 -8889.119} C_VEL
LIN {X 0,Y 440.506,Z 497.625,A -85,B 0,C 180,E1 -8890.024,E2 -8890.024} C_VEL
LIN {X 0,Y 439.524,Z 501.053,A -85,B 0,C 180,E1 -8890.631,E2 -8890.631} C_VEL
LIN {X 0,Y 439.15,Z 506.611,A -85,B 0,C 180,E1 -8891.816,E2 -8891.816} C_VEL
LIN {X 0,Y 438.802,Z 512.042,A -85,B 0,C 180,E1 -8893.244,E2 -8893.244} C_VEL
LIN {X 0,Y 438.599,Z 516.234,A -85,B 0,C 180,E1 -8894.669,E2 -8894.669} C_VEL
LIN {X 0,Y 438.394,Z 519.314,A -85,B 0,C 180,E1 -8896.086,E2 -8896.086} C_VEL
LIN {X 0,Y 438.309,Z 520.813,A -85,B 0,C 180,E1 -8897.027,E2 -8897.027} C_VEL
LIN {X 0,Y 438.336,Z 521.849,A -85,B 0,C 180,E1 -8897.969,E2 -8897.969} C_VEL
LIN {X 0,Y 438.239,Z 522.742,A -85,B 0,C 180,E1 -8899.839,E2 -8899.839} C_VEL
LIN {X 0,Y 438.216,Z 522.568,A -85,B 0,C 180,E1 -8900.771,E2 -8900.771} C_VEL
LIN {X 0,Y 438.329,Z 520.996,A -85,B 0,C 180,E1 -8902.63,E2 -8902.63} C_VEL
LIN {X 0,Y 438.436,Z 519.481,A -85,B 0,C 180,E1 -8903.638,E2 -8903.638} C_VEL
LIN {X 0,Y 438.484,Z 516.734,A -85,B 0,C 180,E1 -8904.942,E2 -8904.942} C_VEL
LIN {X 0,Y 438.661,Z 512.821,A -85,B 0,C 180,E1 -8906.325,E2 -8906.325} C_VEL
LIN {X 0,Y 438.833,Z 507.794,A -85,B 0,C 180,E1 -8907.705,E2 -8907.705} C_VEL
LIN {X 0,Y 439.185,Z 501.466,A -85,B 0,C 180,E1 -8909.083,E2 -8909.083} C_VEL
LIN {X 0,Y 439.685,Z 493.564,A -85,B 0,C 180,E1 -8910.457,E2 -8910.457} C_VEL
LIN {X 0,Y 440.18,Z 483.781,A -85,B 0,C 180,E1 -8911.829,E2 -8911.829} C_VEL
LIN {X 0,Y 440.712,Z 473.533,A -85,B 0,C 180,E1 -8912.97,E2 -8912.97} C_VEL
LIN {X 0,Y 441.464,Z 463.343,A -85,B 0,C 180,E1 -8913.879,E2 -8913.879} C_VEL
LIN {X 0,Y 441.998,Z 452.271,A -85,B 0,C 180,E1 -8914.674,E2 -8914.674} C_VEL
LIN {X 0,Y 442.459,Z 439.911,A -85,B 0,C 180,E1 -8915.354,E2 -8915.354} C_VEL
LIN {X 0,Y 442.753,Z 426.762,A -85,B 0,C 180,E1 -8915.864,E2 -8915.864} C_VEL
LIN {X 0,Y 443.059,Z 413.859,A -85,B 0,C 180,E1 -8916.175,E2 -8916.175} C_VEL
LIN {X 0,Y 443.799,Z 328.671,A -85,B 0,C 180,E1 -8917.556,E2 -8917.556} C_VEL
LIN {X 0,Y 440.539,Z 311.794,A -85,B 0,C 180,E1 -8917.961,E2 -8917.961} C_VEL
LIN {X 0,Y 440.734,Z 303.698,A -85,B 0,C 180,E1 -8919.638,E2 -8919.638} C_VEL
LIN {X 0,Y 439.452,Z 295.746,A -85,B 0,C 180,E1 -8921.414,E2 -8921.414} C_VEL
LIN {X 0,Y 439.417,Z 295.75,A -85,B 0,C 180,E1 -8923.88,E2 -8923.88} C_VEL
LIN {X 0,Y 439.443,Z 295.744,A -85,B 0,C 180,E1 -8926.73,E2 -8926.73} C_VEL
LIN {X 0,Y 439.399,Z 295.747,A -85,B 0,C 180,E1 -8929.626,E2 -8929.626} C_VEL
LIN {X 0,Y 439.36,Z 295.759,A -85,B 0,C 180,E1 -8932.575,E2 -8932.575} C_VEL
LIN {X 0,Y 439.362,Z 295.751,A -85,B 0,C 180,E1 -8935.587,E2 -8935.587} C_VEL
LIN {X 0,Y 439.386,Z 295.757,A -85,B 0,C 180,E1 -8938.675,E2 -8938.675} C_VEL
LIN {X 0,Y 439.364,Z 295.751,A -85,B 0,C 180,E1 -8942.029,E2 -8942.029} C_VEL
LIN {X 0,Y 439.388,Z 295.75,A -85,B 0,C 180,E1 -8945.339,E2 -8945.339} C_VEL
LIN {X 0,Y 439.363,Z 295.755,A -85,B 0,C 180,E1 -8948.596,E2 -8948.596} C_VEL
LIN {X 0,Y 439.362,Z 295.756,A -85,B 0,C 180,E1 -8951.253,E2 -8951.253} C_VEL
LIN {X 0,Y 439.392,Z 295.751,A -85,B 0,C 180,E1 -8954.729,E2 -8954.729} C_VEL
LIN {X 0,Y 439.377,Z 295.75,A -85,B 0,C 180,E1 -8957.794,E2 -8957.794} C_VEL
LIN {X 0,Y 439.382,Z 295.749,A -85,B 0,C 180,E1 -8960.223,E2 -8960.223} C_VEL
LIN {X 0,Y 439.366,Z 295.754,A -85,B 0,C 180,E1 -8963.712,E2 -8963.712} C_VEL
LIN {X 0,Y 439.365,Z 295.754,A -85,B 0,C 180,E1 -8967.053,E2 -8967.053} C_VEL
LIN {X 0,Y 439.373,Z 295.75,A -85,B 0,C 180,E1 -8970.274,E2 -8970.274} C_VEL
LIN {X 0,Y 439.411,Z 295.75,A -85,B 0,C 180,E1 -8973.395,E2 -8973.395} C_VEL
LIN {X 0,Y 439.375,Z 295.75,A -85,B 0,C 180,E1 -8976.429,E2 -8976.429} C_VEL
LIN {X 0,Y 439.379,Z 295.752,A -85,B 0,C 180,E1 -8979.397,E2 -8979.397} C_VEL
LIN {X 0,Y 439.423,Z 295.746,A -85,B 0,C 180,E1 -8982.309,E2 -8982.309} C_VEL
LIN {X 0,Y 439.442,Z 295.742,A -85,B 0,C 180,E1 -8985.174,E2 -8985.174} C_VEL
LIN {X 0,Y 439.475,Z 295.746,A -85,B 0,C 180,E1 -8988.001,E2 -8988.001} C_VEL
LIN {X 0,Y 439.524,Z 295.734,A -85,B 0,C 180,E1 -8991.726,E2 -8991.726} C_VEL
LIN {X 0,Y 439.601,Z 295.725,A -85,B 0,C 180,E1 -8994.496,E2 -8994.496} C_VEL
LIN {X 0,Y 439.626,Z 295.725,A -85,B 0,C 180,E1 -8998.168,E2 -8998.168} C_VEL
LIN {X 0,Y 439.752,Z 295.707,A -85,B 0,C 180,E1 -9000,E2 -9000} C_VEL
LIN {X 0,Y 439.632,Z 295.721,A -85,B 0,C 180,E1 -9002.749,E2 -9002.749} C_VEL
LIN {X 0,Y 439.609,Z 295.728,A -85,B 0,C 180,E1 -9006.425,E2 -9006.425} C_VEL
LIN {X 0,Y 439.493,Z 295.736,A -85,B 0,C 180,E1 -9009.202,E2 -9009.202} C_VEL
LIN {X 0,Y 439.457,Z 295.744,A -85,B 0,C 180,E1 -9012.938,E2 -9012.938} C_VEL
LIN {X 0,Y 439.439,Z 295.745,A -85,B 0,C 180,E1 -9016.349,E2 -9016.349} C_VEL
LIN {X 0,Y 439.395,Z 295.747,A -85,B 0,C 180,E1 -9019.627,E2 -9019.627} C_VEL
LIN {X 0,Y 439.357,Z 295.755,A -85,B 0,C 180,E1 -9022.576,E2 -9022.576} C_VEL
LIN {X 0,Y 439.399,Z 295.748,A -85,B 0,C 180,E1 -9025.585,E2 -9025.585} C_VEL
LIN {X 0,Y 439.419,Z 295.747,A -85,B 0,C 180,E1 -9028.674,E2 -9028.674} C_VEL
LIN {X 0,Y 439.379,Z 295.749,A -85,B 0,C 180,E1 -9032.034,E2 -9032.034} C_VEL
LIN {X 0,Y 439.39,Z 295.755,A -85,B 0,C 180,E1 -9035.341,E2 -9035.341} C_VEL
LIN {X 0,Y 439.385,Z 295.749,A -85,B 0,C 180,E1 -9038.595,E2 -9038.595} C_VEL
LIN {X 0,Y 439.385,Z 295.754,A -85,B 0,C 180,E1 -9041.258,E2 -9041.258} C_VEL
LIN {X 0,Y 439.401,Z 295.747,A -85,B 0,C 180,E1 -9044.73,E2 -9044.73} C_VEL
LIN {X 0,Y 439.392,Z 295.753,A -85,B 0,C 180,E1 -9047.797,E2 -9047.797} C_VEL
LIN {X 0,Y 439.391,Z 295.749,A -85,B 0,C 180,E1 -9050.225,E2 -9050.225} C_VEL
LIN {X 0,Y 439.371,Z 295.758,A -85,B 0,C 180,E1 -9053.714,E2 -9053.714} C_VEL
LIN {X 0,Y 439.37,Z 295.75,A -85,B 0,C 180,E1 -9057.055,E2 -9057.055} C_VEL
LIN {X 0,Y 439.381,Z 295.755,A -85,B 0,C 180,E1 -9060.275,E2 -9060.275} C_VEL
LIN {X 0,Y 439.464,Z 295.807,A -85,B 0,C 180,E1 -9063.335,E2 -9063.335} C_VEL
LIN {X 0,Y 441.858,Z 308.378,A -85,B 0,C 180,E1 -9065.823,E2 -9065.823} C_VEL
LIN {X 0,Y 441.357,Z 320.346,A -85,B 0,C 180,E1 -9068.026,E2 -9068.026} C_VEL
LIN {X 0,Y 440.452,Z 338.862,A -85,B 0,C 180,E1 -9071.391,E2 -9071.391} C_VEL
LIN {X 0,Y 440.269,Z 342.605,A -85,B 0,C 180,E1 -9072.056,E2 -9072.056} C_VEL
LIN {X 0,Y 443.652,Z 366.177,A -85,B 0,C 180,E1 -9072.567,E2 -9072.567} C_VEL
LIN {X 0,Y 442.849,Z 451.296,A -85,B 0,C 180,E1 -9073.965,E2 -9073.965} C_VEL
LIN {X 0,Y 442.419,Z 464.502,A -85,B 0,C 180,E1 -9074.363,E2 -9074.363} C_VEL
LIN {X 0,Y 441.944,Z 476.657,A -85,B 0,C 180,E1 -9074.907,E2 -9074.907} C_VEL
LIN {X 0,Y 441.402,Z 488.113,A -85,B 0,C 180,E1 -9075.595,E2 -9075.595} C_VEL
LIN {X 0,Y 440.782,Z 499.647,A -85,B 0,C 180,E1 -9076.494,E2 -9076.494} C_VEL
LIN {X 0,Y 440.164,Z 510.456,A -85,B 0,C 180,E1 -9077.553,E2 -9077.553} C_VEL
LIN {X 0,Y 439.661,Z 519.974,A -85,B 0,C 180,E1 -9078.708,E2 -9078.708} C_VEL
LIN {X 0,Y 439.112,Z 529.129,A -85,B 0,C 180,E1 -9080.093,E2 -9080.093} C_VEL
LIN {X 0,Y 438.781,Z 536.507,A -85,B 0,C 180,E1 -9081.48,E2 -9081.48} C_VEL
LIN {X 0,Y 438.536,Z 541.5,A -85,B 0,C 180,E1 -9082.635,E2 -9082.635} C_VEL
LIN {X 0,Y 438.358,Z 546.321,A -85,B 0,C 180,E1 -9084.011,E2 -9084.011} C_VEL
LIN {X 0,Y 438.341,Z 550.062,A -85,B 0,C 180,E1 -9085.402,E2 -9085.402} C_VEL
LIN {X 0,Y 438.285,Z 551.977,A -85,B 0,C 180,E1 -9086.323,E2 -9086.323} C_VEL
LIN {X 0,Y 438.359,Z 553.451,A -85,B 0,C 180,E1 -9087.244,E2 -9087.244} C_VEL
LIN {X 0,Y 438.278,Z 555.126,A -85,B 0,C 180,E1 -9089.082,E2 -9089.082} C_VEL
LIN {X 0,Y 438.281,Z 555.382,A -85,B 0,C 180,E1 -9090,E2 -9090} C_VEL
LIN {X 0,Y 438.254,Z 555.227,A -85,B 0,C 180,E1 -9090.919,E2 -9090.919} C_VEL
LIN {X 0,Y 438.295,Z 554.652,A -85,B 0,C 180,E1 -9091.838,E2 -9091.838} C_VEL
LIN {X 0,Y 438.341,Z 553.689,A -85,B 0,C 180,E1 -9092.757,E2 -9092.757} C_VEL
LIN {X 0,Y 438.282,Z 552.327,A -85,B 0,C 180,E1 -9093.678,E2 -9093.678} C_VEL
LIN {X 0,Y 438.383,Z 549.46,A -85,B 0,C 180,E1 -9095.059,E2 -9095.059} C_VEL
LIN {X 0,Y 438.449,Z 545.566,A -85,B 0,C 180,E1 -9096.443,E2 -9096.443} C_VEL
LIN {X 0,Y 438.65,Z 540.553,A -85,B 0,C 180,E1 -9097.828,E2 -9097.828} C_VEL
LIN {X 0,Y 438.957,Z 534.268,A -85,B 0,C 180,E1 -9099.213,E2 -9099.213} C_VEL
LIN {X 0,Y 439.386,Z 526.418,A -85,B 0,C 180,E1 -9100.6,E2 -9100.6} C_VEL
LIN {X 0,Y 440.108,Z 516.651,A -85,B 0,C 180,E1 -9101.982,E2 -9101.982} C_VEL
LIN {X 0,Y 440.751,Z 507.032,A -85,B 0,C 180,E1 -9103.083,E2 -9103.083} C_VEL
LIN {X 0,Y 441.335,Z 496.528,A -85,B 0,C 180,E1 -9104.055,E2 -9104.055} C_VEL
LIN {X 0,Y 442.104,Z 483.896,A -85,B 0,C 180,E1 -9104.971,E2 -9104.971} C_VEL
LIN {X 0,Y 442.775,Z 471.302,A -85,B 0,C 180,E1 -9105.655,E2 -9105.655} C_VEL
LIN {X 0,Y 443.347,Z 457.838,A -85,B 0,C 180,E1 -9106.165,E2 -9106.165} C_VEL
LIN {X 0,Y 443.647,Z 444.44,A -85,B 0,C 180,E1 -9106.479,E2 -9106.479} C_VEL
LIN {X 0,Y 444.471,Z 366.162,A -85,B 0,C 180,E1 -9107.759,E2 -9107.759} C_VEL
LIN {X 0,Y 441.275,Z 346.038,A -85,B 0,C 180,E1 -9108.251,E2 -9108.251} C_VEL
LIN {X 0,Y 440.596,Z 342.155,A -85,B 0,C 180,E1 -9108.369,E2 -9108.369} C_VEL
LIN {X 0,Y 441.626,Z 323.984,A -85,B 0,C 180,E1 -9111.716,E2 -9111.716} C_VEL
LIN {X 0,Y 442.382,Z 310.987,A -85,B 0,C 180,E1 -9114.147,E2 -9114.147} C_VEL
LIN {X 0,Y 440.808,Z 301.881,A -85,B 0,C 180,E1 -9116.005,E2 -9116.005} C_VEL
LIN {X 0,Y 439.447,Z 295.75,A -85,B 0,C 180,E1 -9117.309,E2 -9117.309} C_VEL
LIN {X 0,Y 439.363,Z 295.757,A -85,B 0,C 180,E1 -9120.788,E2 -9120.788} C_VEL
LIN {X 0,Y 439.389,Z 295.754,A -85,B 0,C 180,E1 -9124.044,E2 -9124.044} C_VEL
LIN {X 0,Y 439.35,Z 295.757,A -85,B 0,C 180,E1 -9126.887,E2 -9126.887} C_VEL
LIN {X 0,Y 439.403,Z 295.75,A -85,B 0,C 180,E1 -9129.849,E2 -9129.849} C_VEL
LIN {X 0,Y 439.383,Z 295.755,A -85,B 0,C 180,E1 -9132.627,E2 -9132.627} C_VEL
LIN {X 0,Y 439.4,Z 295.749,A -85,B 0,C 180,E1 -9135.27,E2 -9135.27} C_VEL
LIN {X 0,Y 439.389,Z 295.755,A -85,B 0,C 180,E1 -9138.743,E2 -9138.743} C_VEL
LIN {X 0,Y 439.373,Z 295.751,A -85,B 0,C 180,E1 -9141.608,E2 -9141.608} C_VEL
LIN {X 0,Y 439.399,Z 295.754,A -85,B 0,C 180,E1 -9144.844,E2 -9144.844} C_VEL
LIN {X 0,Y 439.372,Z 295.751,A -85,B 0,C 180,E1 -9148.139,E2 -9148.139} C_VEL
LIN {X 0,Y 439.432,Z 295.745,A -85,B 0,C 180,E1 -9151.598,E2 -9151.598} C_VEL
LIN {X 0,Y 439.4,Z 295.747,A -85,B 0,C 180,E1 -9154.415,E2 -9154.415} C_VEL
LIN {X 0,Y 439.364,Z 295.755,A -85,B 0,C 180,E1 -9157.424,E2 -9157.424} C_VEL
LIN {X 0,Y 439.441,Z 295.741,A -85,B 0,C 180,E1 -9160.663,E2 -9160.663} C_VEL
LIN {X 0,Y 439.462,Z 295.738,A -85,B 0,C 180,E1 -9164.224,E2 -9164.224} C_VEL
LIN {X 0,Y 439.482,Z 295.738,A -85,B 0,C 180,E1 -9168.001,E2 -9168.001} C_VEL
LIN {X 0,Y 439.547,Z 295.732,A -85,B 0,C 180,E1 -9171.726,E2 -9171.726} C_VEL
LIN {X 0,Y 439.619,Z 295.714,A -85,B 0,C 180,E1 -9174.496,E2 -9174.496} C_VEL
LIN {X 0,Y 439.632,Z 295.715,A -85,B 0,C 180,E1 -9178.168,E2 -9178.168} C_VEL
LIN {X 0,Y 439.76,Z 295.703,A -85,B 0,C 180,E1 -9180,E2 -9180} C_VEL
LIN {X 0,Y 439.639,Z 295.712,A -85,B 0,C 180,E1 -9182.749,E2 -9182.749} C_VEL
LIN {X 0,Y 439.611,Z 295.722,A -85,B 0,C 180,E1 -9186.425,E2 -9186.425} C_VEL
LIN {X 0,Y 439.498,Z 295.733,A -85,B 0,C 180,E1 -9189.202,E2 -9189.202} C_VEL
LIN {X 0,Y 439.464,Z 295.74,A -85,B 0,C 180,E1 -9192.938,E2 -9192.938} C_VEL
LIN {X 0,Y 439.446,Z 295.744,A -85,B 0,C 180,E1 -9196.349,E2 -9196.349} C_VEL
LIN {X 0,Y 439.401,Z 295.746,A -85,B 0,C 180,E1 -9199.626,E2 -9199.626} C_VEL
LIN {X 0,Y 439.364,Z 295.757,A -85,B 0,C 180,E1 -9202.575,E2 -9202.575} C_VEL
LIN {X 0,Y 439.404,Z 295.746,A -85,B 0,C 180,E1 -9205.585,E2 -9205.585} C_VEL
LIN {X 0,Y 439.416,Z 295.746,A -85,B 0,C 180,E1 -9208.673,E2 -9208.673} C_VEL
LIN {X 0,Y 439.368,Z 295.748,A -85,B 0,C 180,E1 -9212.03,E2 -9212.03} C_VEL
LIN {X 0,Y 439.393,Z 295.753,A -85,B 0,C 180,E1 -9215.34,E2 -9215.34} C_VEL
LIN {X 0,Y 439.376,Z 295.751,A -85,B 0,C 180,E1 -9218.596,E2 -9218.596} C_VEL
LIN {X 0,Y 439.388,Z 295.755,A -85,B 0,C 180,E1 -9221.257,E2 -9221.257} C_VEL
LIN {X 0,Y 439.399,Z 295.749,A -85,B 0,C 180,E1 -9224.73,E2 -9224.73} C_VEL
LIN {X 0,Y 439.395,Z 295.752,A -85,B 0,C 180,E1 -9227.796,E2 -9227.796} C_VEL
LIN {X 0,Y 439.395,Z 295.752,A -85,B 0,C 180,E1 -9230.224,E2 -9230.224} C_VEL
LIN {X 0,Y 439.374,Z 295.758,A -85,B 0,C 180,E1 -9233.713,E2 -9233.713} C_VEL
LIN {X 0,Y 439.376,Z 295.755,A -85,B 0,C 180,E1 -9237.054,E2 -9237.054} C_VEL
LIN {X 0,Y 439.416,Z 295.804,A -85,B 0,C 180,E1 -9238.244,E2 -9238.244} C_VEL
LIN {X 0,Y 441.051,Z 304.305,A -85,B 0,C 180,E1 -9240.14,E2 -9240.14} C_VEL
LIN {X 0,Y 440.962,Z 312.108,A -85,B 0,C 180,E1 -9241.715,E2 -9241.715} C_VEL
LIN {X 0,Y 444.776,Z 329.759,A -85,B 0,C 180,E1 -9242.201,E2 -9242.201} C_VEL
LIN {X 0,Y 443.719,Z 418.826,A -85,B 0,C 180,E1 -9243.673,E2 -9243.673} C_VEL
LIN {X 0,Y 443.311,Z 431.812,A -85,B 0,C 180,E1 -9244.058,E2 -9244.058} C_VEL
LIN {X 0,Y 442.971,Z 444.574,A -85,B 0,C 180,E1 -9244.636,E2 -9244.636} C_VEL
LIN {X 0,Y 442.451,Z 455.458,A -85,B 0,C 180,E1 -9245.292,E2 -9245.292} C_VEL
LIN {X 0,Y 441.773,Z 467.042,A -85,B 0,C 180,E1 -9246.191,E2 -9246.191} C_VEL
LIN {X 0,Y 441.095,Z 477.988,A -85,B 0,C 180,E1 -9247.271,E2 -9247.271} C_VEL
LIN {X 0,Y 440.405,Z 487.764,A -85,B 0,C 180,E1 -9248.467,E2 -9248.467} C_VEL
LIN {X 0,Y 439.819,Z 497.079,A -85,B 0,C 180,E1 -9249.906,E2 -9249.906} C_VEL
LIN {X 0,Y 439.524,Z 501.053,A -85,B 0,C 180,E1 -9250.631,E2 -9250.631} C_VEL
LIN {X 0,Y 438.57,Z 504.322,A -85,B 0,C 180,E1 -9251.263,E2 -9251.263} C_VEL
LIN {X 0,Y 435.407,Z 509.199,A -85,B 0,C 180,E1 -9252.318,E2 -9252.318} C_VEL
LIN {X 0,Y 432.356,Z 513.352,A -85,B 0,C 180,E1 -9253.438,E2 -9253.438} C_VEL
LIN {X 0,Y 431.587,Z 515.483,A -85,B 0,C 180,E1 -9254.162,E2 -9254.162} C_VEL
LIN {X 0,Y 431.331,Z 519.326,A -85,B 0,C 180,E1 -9255.853,E2 -9255.853} C_VEL
LIN {X 0,Y 431.244,Z 520.894,A -85,B 0,C 180,E1 -9256.811,E2 -9256.811} C_VEL
LIN {X 0,Y 431.254,Z 522.116,A -85,B 0,C 180,E1 -9257.905,E2 -9257.905} C_VEL
LIN {X 0,Y 431.146,Z 522.985,A -85,B 0,C 180,E1 -9259.67,E2 -9259.67} C_VEL
LIN {X 0,Y 431.119,Z 522.89,A -85,B 0,C 180,E1 -9260.618,E2 -9260.618} C_VEL
LIN {X 0,Y 431.158,Z 522.356,A -85,B 0,C 180,E1 -9261.564,E2 -9261.564} C_VEL
LIN {X 0,Y 431.239,Z 521.42,A -85,B 0,C 180,E1 -9262.508,E2 -9262.508} C_VEL
LIN {X 0,Y 431.357,Z 519.779,A -85,B 0,C 180,E1 -9263.646,E2 -9263.646} C_VEL
LIN {X 0,Y 431.387,Z 516.147,A -85,B 0,C 180,E1 -9265.327,E2 -9265.327} C_VEL
LIN {X 0,Y 431.626,Z 511.97,A -85,B 0,C 180,E1 -9266.733,E2 -9266.733} C_VEL
LIN {X 0,Y 431.922,Z 505.636,A -85,B 0,C 180,E1 -9268.368,E2 -9268.368} C_VEL
LIN {X 0,Y 432.4,Z 498.727,A -85,B 0,C 180,E1 -9269.767,E2 -9269.767} C_VEL
LIN {X 0,Y 432.918,Z 490.091,A -85,B 0,C 180,E1 -9271.162,E2 -9271.162} C_VEL
LIN {X 0,Y 433.322,Z 481.285,A -85,B 0,C 180,E1 -9272.323,E2 -9272.323} C_VEL
LIN {X 0,Y 433.938,Z 471.585,A -85,B 0,C 180,E1 -9273.365,E2 -9273.365} C_VEL
LIN {X 0,Y 434.721,Z 460.891,A -85,B 0,C 180,E1 -9274.288,E2 -9274.288} C_VEL
LIN {X 0,Y 435.221,Z 448.988,A -85,B 0,C 180,E1 -9275.095,E2 -9275.095} C_VEL
LIN {X 0,Y 435.679,Z 436.583,A -85,B 0,C 180,E1 -9275.728,E2 -9275.728} C_VEL
LIN {X 0,Y 435.895,Z 426.48,A -85,B 0,C 180,E1 -9276.102,E2 -9276.102} C_VEL
LIN {X 0,Y 436.203,Z 413.194,A -85,B 0,C 180,E1 -9276.417,E2 -9276.417} C_VEL
LIN {X 0,Y 437.027,Z 329.921,A -85,B 0,C 180,E1 -9277.784,E2 -9277.784} C_VEL
LIN {X 0,Y 433.623,Z 311.942,A -85,B 0,C 180,E1 -9278.237,E2 -9278.237} C_VEL
LIN {X 0,Y 433.747,Z 304.531,A -85,B 0,C 180,E1 -9279.795,E2 -9279.795} C_VEL
LIN {X 0,Y 432.418,Z 296.622,A -85,B 0,C 180,E1 -9281.573,E2 -9281.573} C_VEL
LIN {X 0,Y 432.366,Z 296.629,A -85,B 0,C 180,E1 -9284.111,E2 -9284.111} C_VEL
LIN {X 0,Y 432.385,Z 296.621,A -85,B 0,C 180,E1 -9287.011,E2 -9287.011} C_VEL
LIN {X 0,Y 432.336,Z 296.629,A -85,B 0,C 180,E1 -9289.96,E2 -9289.96} C_VEL
LIN {X 0,Y 432.307,Z 296.633,A -85,B 0,C 180,E1 -9292.964,E2 -9292.964} C_VEL
LIN {X 0,Y 432.313,Z 296.631,A -85,B 0,C 180,E1 -9296.035,E2 -9296.035} C_VEL
LIN {X 0,Y 432.322,Z 296.63,A -85,B 0,C 180,E1 -9299.188,E2 -9299.188} C_VEL
LIN {X 0,Y 432.318,Z 296.632,A -85,B 0,C 180,E1 -9302.442,E2 -9302.442} C_VEL
LIN {X 0,Y 432.339,Z 296.626,A -85,B 0,C 180,E1 -9305.631,E2 -9305.631} C_VEL
LIN {X 0,Y 432.325,Z 296.633,A -85,B 0,C 180,E1 -9308.712,E2 -9308.712} C_VEL
LIN {X 0,Y 432.303,Z 296.631,A -85,B 0,C 180,E1 -9311.799,E2 -9311.799} C_VEL
LIN {X 0,Y 432.327,Z 296.628,A -85,B 0,C 180,E1 -9314.347,E2 -9314.347} C_VEL
LIN {X 0,Y 432.31,Z 296.636,A -85,B 0,C 180,E1 -9317.016,E2 -9317.016} C_VEL
LIN {X 0,Y 432.307,Z 296.631,A -85,B 0,C 180,E1 -9319.823,E2 -9319.823} C_VEL
LIN {X 0,Y 432.298,Z 296.635,A -85,B 0,C 180,E1 -9323.021,E2 -9323.021} C_VEL
LIN {X 0,Y 432.352,Z 296.626,A -85,B 0,C 180,E1 -9325.996,E2 -9325.996} C_VEL
LIN {X 0,Y 432.339,Z 296.634,A -85,B 0,C 180,E1 -9329.489,E2 -9329.489} C_VEL
LIN {X 0,Y 432.377,Z 296.622,A -85,B 0,C 180,E1 -9332.927,E2 -9332.927} C_VEL
LIN {X 0,Y 432.359,Z 296.627,A -85,B 0,C 180,E1 -9336.023,E2 -9336.023} C_VEL
LIN {X 0,Y 432.341,Z 296.626,A -85,B 0,C 180,E1 -9339.046,E2 -9339.046} C_VEL
LIN {X 0,Y 432.37,Z 296.628,A -85,B 0,C 180,E1 -9342.011,E2 -9342.011} C_VEL
LIN {X 0,Y 432.392,Z 296.619,A -85,B 0,C 180,E1 -9344.926,E2 -9344.926} C_VEL
LIN {X 0,Y 432.45,Z 296.618,A -85,B 0,C 180,E1 -9347.803,E2 -9347.803} C_VEL
LIN {X 0,Y 432.474,Z 296.611,A -85,B 0,C 180,E1 -9351.59,E2 -9351.59} C_VEL
LIN {X 0,Y 432.576,Z 296.601,A -85,B 0,C 180,E1 -9354.406,E2 -9354.406} C_VEL
LIN {X 0,Y 432.596,Z 296.601,A -85,B 0,C 180,E1 -9358.138,E2 -9358.138} C_VEL
LIN {X 0,Y 432.722,Z 296.582,A -85,B 0,C 180,E1 -9360,E2 -9360} C_VEL
LIN {X 0,Y 432.584,Z 296.599,A -85,B 0,C 180,E1 -9362.794,E2 -9362.794} C_VEL
LIN {X 0,Y 432.564,Z 296.606,A -85,B 0,C 180,E1 -9366.531,E2 -9366.531} C_VEL
LIN {X 0,Y 432.436,Z 296.614,A -85,B 0,C 180,E1 -9369.353,E2 -9369.353} C_VEL
LIN {X 0,Y 432.423,Z 296.622,A -85,B 0,C 180,E1 -9372.804,E2 -9372.804} C_VEL
LIN {X 0,Y 432.405,Z 296.622,A -85,B 0,C 180,E1 -9376.479,E2 -9376.479} C_VEL
LIN {X 0,Y 432.331,Z 296.627,A -85,B 0,C 180,E1 -9379.961,E2 -9379.961} C_VEL
LIN {X 0,Y 432.312,Z 296.637,A -85,B 0,C 180,E1 -9382.965,E2 -9382.965} C_VEL
LIN {X 0,Y 432.358,Z 296.624,A -85,B 0,C 180,E1 -9386.033,E2 -9386.033} C_VEL
LIN {X 0,Y 432.346,Z 296.632,A -85,B 0,C 180,E1 -9389.187,E2 -9389.187} C_VEL
LIN {X 0,Y 432.327,Z 296.628,A -85,B 0,C 180,E1 -9392.296,E2 -9392.296} C_VEL
LIN {X 0,Y 432.335,Z 296.628,A -85,B 0,C 180,E1 -9394.678,E2 -9394.678} C_VEL
LIN {X 0,Y 432.342,Z 296.626,A -85,B 0,C 180,E1 -9398.15,E2 -9398.15} C_VEL
LIN {X 0,Y 432.33,Z 296.633,A -85,B 0,C 180,E1 -9401.603,E2 -9401.603} C_VEL
LIN {X 0,Y 432.336,Z 296.626,A -85,B 0,C 180,E1 -9404.347,E2 -9404.347} C_VEL
LIN {X 0,Y 432.316,Z 296.63,A -85,B 0,C 180,E1 -9407.017,E2 -9407.017} C_VEL
LIN {X 0,Y 432.33,Z 296.633,A -85,B 0,C 180,E1 -9409.822,E2 -9409.822} C_VEL
LIN {X 0,Y 432.303,Z 296.631,A -85,B 0,C 180,E1 -9413.023,E2 -9413.023} C_VEL
LIN {X 0,Y 432.357,Z 296.629,A -85,B 0,C 180,E1 -9415.997,E2 -9415.997} C_VEL
LIN {X 0,Y 432.346,Z 296.628,A -85,B 0,C 180,E1 -9419.491,E2 -9419.491} C_VEL
LIN {X 0,Y 432.455,Z 296.616,A -85,B 0,C 180,E1 -9423.096,E2 -9423.096} C_VEL
LIN {X 0,Y 434.838,Z 309.206,A -85,B 0,C 180,E1 -9425.662,E2 -9425.662} C_VEL
LIN {X 0,Y 434.605,Z 317.204,A -85,B 0,C 180,E1 -9427.164,E2 -9427.164} C_VEL
LIN {X 0,Y 433.697,Z 334.433,A -85,B 0,C 180,E1 -9430.352,E2 -9430.352} C_VEL
LIN {X 0,Y 433.312,Z 342.229,A -85,B 0,C 180,E1 -9431.785,E2 -9431.785} C_VEL
LIN {X 0,Y 436.795,Z 366.757,A -85,B 0,C 180,E1 -9432.334,E2 -9432.334} C_VEL
LIN {X 0,Y 435.978,Z 450.853,A -85,B 0,C 180,E1 -9433.735,E2 -9433.735} C_VEL
LIN {X 0,Y 435.532,Z 464.122,A -85,B 0,C 180,E1 -9434.139,E2 -9434.139} C_VEL
LIN {X 0,Y 435.004,Z 476.879,A -85,B 0,C 180,E1 -9434.72,E2 -9434.72} C_VEL
LIN {X 0,Y 434.396,Z 488.999,A -85,B 0,C 180,E1 -9435.478,E2 -9435.478} C_VEL
LIN {X 0,Y 433.766,Z 499.974,A -85,B 0,C 180,E1 -9436.36,E2 -9436.36} C_VEL
LIN {X 0,Y 433.116,Z 510.967,A -85,B 0,C 180,E1 -9437.466,E2 -9437.466} C_VEL
LIN {X 0,Y 432.645,Z 519.474,A -85,B 0,C 180,E1 -9438.523,E2 -9438.523} C_VEL
LIN {X 0,Y 432.05,Z 528.678,A -85,B 0,C 180,E1 -9439.93,E2 -9439.93} C_VEL
LIN {X 0,Y 431.716,Z 536.092,A -85,B 0,C 180,E1 -9441.34,E2 -9441.34} C_VEL
LIN {X 0,Y 431.417,Z 542.887,A -85,B 0,C 180,E1 -9442.983,E2 -9442.983} C_VEL
LIN {X 0,Y 431.274,Z 547.366,A -85,B 0,C 180,E1 -9444.389,E2 -9444.389} C_VEL
LIN {X 0,Y 431.27,Z 549.729,A -85,B 0,C 180,E1 -9445.327,E2 -9445.327} C_VEL
LIN {X 0,Y 431.191,Z 551.655,A -85,B 0,C 180,E1 -9446.262,E2 -9446.262} C_VEL
LIN {X 0,Y 431.268,Z 553.151,A -85,B 0,C 180,E1 -9447.198,E2 -9447.198} C_VEL
LIN {X 0,Y 431.193,Z 554.846,A -85,B 0,C 180,E1 -9449.067,E2 -9449.067} C_VEL
LIN {X 0,Y 431.193,Z 555.112,A -85,B 0,C 180,E1 -9450,E2 -9450} C_VEL
LIN {X 0,Y 431.171,Z 554.977,A -85,B 0,C 180,E1 -9450.934,E2 -9450.934} C_VEL
LIN {X 0,Y 431.219,Z 554.413,A -85,B 0,C 180,E1 -9451.868,E2 -9451.868} C_VEL
LIN {X 0,Y 431.237,Z 553.458,A -85,B 0,C 180,E1 -9452.803,E2 -9452.803} C_VEL
LIN {X 0,Y 431.188,Z 552.108,A -85,B 0,C 180,E1 -9453.739,E2 -9453.739} C_VEL
LIN {X 0,Y 431.294,Z 549.263,A -85,B 0,C 180,E1 -9455.142,E2 -9455.142} C_VEL
LIN {X 0,Y 431.377,Z 545.394,A -85,B 0,C 180,E1 -9456.549,E2 -9456.549} C_VEL
LIN {X 0,Y 431.576,Z 540.407,A -85,B 0,C 180,E1 -9457.957,E2 -9457.957} C_VEL
LIN {X 0,Y 431.921,Z 534.154,A -85,B 0,C 180,E1 -9459.365,E2 -9459.365} C_VEL
LIN {X 0,Y 432.389,Z 526.357,A -85,B 0,C 180,E1 -9460.773,E2 -9460.773} C_VEL
LIN {X 0,Y 433.138,Z 516.636,A -85,B 0,C 180,E1 -9462.177,E2 -9462.177} C_VEL
LIN {X 0,Y 433.78,Z 507.428,A -85,B 0,C 180,E1 -9463.258,E2 -9463.258} C_VEL
LIN {X 0,Y 434.442,Z 496.676,A -85,B 0,C 180,E1 -9464.283,E2 -9464.283} C_VEL
LIN {X 0,Y 435.248,Z 484.15,A -85,B 0,C 180,E1 -9465.212,E2 -9465.212} C_VEL
LIN {X 0,Y 435.975,Z 471.798,A -85,B 0,C 180,E1 -9465.905,E2 -9465.905} C_VEL
LIN {X 0,Y 436.547,Z 458.666,A -85,B 0,C 180,E1 -9466.424,E2 -9466.424} C_VEL
LIN {X 0,Y 436.906,Z 446.032,A -85,B 0,C 180,E1 -9466.741,E2 -9466.741} C_VEL
LIN {X 0,Y 437.73,Z 366.513,A -85,B 0,C 180,E1 -9468.069,E2 -9468.069} C_VEL
LIN {X 0,Y 434.484,Z 346.317,A -85,B 0,C 180,E1 -9468.577,E2 -9468.577} C_VEL
LIN {X 0,Y 433.697,Z 341.988,A -85,B 0,C 180,E1 -9468.692,E2 -9468.692} C_VEL
LIN {X 0,Y 434.868,Z 322.635,A -85,B 0,C 180,E1 -9472.321,E2 -9472.321} C_VEL
LIN {X 0,Y 435.487,Z 312.246,A -85,B 0,C 180,E1 -9474.301,E2 -9474.301} C_VEL
LIN {X 0,Y 433.643,Z 302.135,A -85,B 0,C 180,E1 -9476.411,E2 -9476.411} C_VEL
LIN {X 0,Y 432.43,Z 296.625,A -85,B 0,C 180,E1 -9477.626,E2 -9477.626} C_VEL
LIN {X 0,Y 432.323,Z 296.635,A -85,B 0,C 180,E1 -9481.346,E2 -9481.346} C_VEL
LIN {X 0,Y 432.342,Z 296.631,A -85,B 0,C 180,E1 -9484.677,E2 -9484.677} C_VEL
LIN {X 0,Y 432.336,Z 296.633,A -85,B 0,C 180,E1 -9488.15,E2 -9488.15} C_VEL
LIN {X 0,Y 432.333,Z 296.629,A -85,B 0,C 180,E1 -9491.602,E2 -9491.602} C_VEL
LIN {X 0,Y 432.334,Z 296.633,A -85,B 0,C 180,E1 -9494.347,E2 -9494.347} C_VEL
LIN {X 0,Y 432.321,Z 296.632,A -85,B 0,C 180,E1 -9497.015,E2 -9497.015} C_VEL
LIN {X 0,Y 432.333,Z 296.625,A -85,B 0,C 180,E1 -9499.821,E2 -9499.821} C_VEL
LIN {X 0,Y 432.306,Z 296.634,A -85,B 0,C 180,E1 -9503.022,E2 -9503.022} C_VEL
LIN {X 0,Y 432.359,Z 296.621,A -85,B 0,C 180,E1 -9505.996,E2 -9505.996} C_VEL
LIN {X 0,Y 432.347,Z 296.626,A -85,B 0,C 180,E1 -9509.489,E2 -9509.489} C_VEL
LIN {X 0,Y 432.39,Z 296.624,A -85,B 0,C 180,E1 -9512.928,E2 -9512.928} C_VEL
LIN {X 0,Y 432.369,Z 296.623,A -85,B 0,C 180,E1 -9516.023,E2 -9516.023} C_VEL
LIN {X 0,Y 432.35,Z 296.629,A -85,B 0,C 180,E1 -9519.046,E2 -9519.046} C_VEL
LIN {X 0,Y 432.377,Z 296.622,A -85,B 0,C 180,E1 -9522.011,E2 -9522.011} C_VEL
LIN {X 0,Y 432.395,Z 296.619,A -85,B 0,C 180,E1 -9524.926,E2 -9524.926} C_VEL
LIN {X 0,Y 432.458,Z 296.615,A -85,B 0,C 180,E1 -9527.803,E2 -9527.803} C_VEL
LIN {X 0,Y 432.491,Z 296.609,A -85,B 0,C 180,E1 -9531.59,E2 -9531.59} C_VEL
LIN {X 0,Y 432.595,Z 296.59,A -85,B 0,C 180,E1 -9534.406,E2 -9534.406} C_VEL
LIN {X 0,Y 432.602,Z 296.591,A -85,B 0,C 180,E1 -9538.138,E2 -9538.138} C_VEL
LIN {X 0,Y 432.73,Z 296.578,A -85,B 0,C 180,E1 -9540,E2 -9540} C_VEL
LIN {X 0,Y 432.591,Z 296.59,A -85,B 0,C 180,E1 -9542.794,E2 -9542.794} C_VEL
LIN {X 0,Y 432.567,Z 296.598,A -85,B 0,C 180,E1 -9546.53,E2 -9546.53} C_VEL
LIN {X 0,Y 432.441,Z 296.612,A -85,B 0,C 180,E1 -9549.353,E2 -9549.353} C_VEL
LIN {X 0,Y 432.429,Z 296.617,A -85,B 0,C 180,E1 -9552.803,E2 -9552.803} C_VEL
LIN {X 0,Y 432.411,Z 296.62,A -85,B 0,C 180,E1 -9556.479,E2 -9556.479} C_VEL
LIN {X 0,Y 432.337,Z 296.627,A -85,B 0,C 180,E1 -9559.96,E2 -9559.96} C_VEL
LIN {X 0,Y 432.318,Z 296.633,A -85,B 0,C 180,E1 -9562.964,E2 -9562.964} C_VEL
LIN {X 0,Y 432.363,Z 296.623,A -85,B 0,C 180,E1 -9566.032,E2 -9566.032} C_VEL
LIN {X 0,Y 432.342,Z 296.63,A -85,B 0,C 180,E1 -9569.187,E2 -9569.187} C_VEL
LIN {X 0,Y 432.322,Z 296.627,A -85,B 0,C 180,E1 -9572.443,E2 -9572.443} C_VEL
LIN {X 0,Y 432.343,Z 296.628,A -85,B 0,C 180,E1 -9575.632,E2 -9575.632} C_VEL
LIN {X 0,Y 432.339,Z 296.628,A -85,B 0,C 180,E1 -9578.714,E2 -9578.714} C_VEL
LIN {X 0,Y 432.333,Z 296.63,A -85,B 0,C 180,E1 -9581.797,E2 -9581.797} C_VEL
LIN {X 0,Y 432.333,Z 296.628,A -85,B 0,C 180,E1 -9584.347,E2 -9584.347} C_VEL
LIN {X 0,Y 432.319,Z 296.632,A -85,B 0,C 180,E1 -9587.016,E2 -9587.016} C_VEL
LIN {X 0,Y 432.333,Z 296.633,A -85,B 0,C 180,E1 -9589.821,E2 -9589.821} C_VEL
LIN {X 0,Y 432.306,Z 296.633,A -85,B 0,C 180,E1 -9593.022,E2 -9593.022} C_VEL
LIN {X 0,Y 432.36,Z 296.631,A -85,B 0,C 180,E1 -9595.997,E2 -9595.997} C_VEL
LIN {X 0,Y 432.353,Z 296.664,A -85,B 0,C 180,E1 -9597.959,E2 -9597.959} C_VEL
LIN {X 0,Y 434.049,Z 305.063,A -85,B 0,C 180,E1 -9599.871,E2 -9599.871} C_VEL
LIN {X 0,Y 434.121,Z 310.144,A -85,B 0,C 180,E1 -9600.951,E2 -9600.951} C_VEL
LIN {X 0,Y 434.081,Z 312.033,A -85,B 0,C 180,E1 -9601.346,E2 -9601.346} C_VEL
LIN {X 0,Y 438.095,Z 330.739,A -85,B 0,C 180,E1 -9601.894,E2 -9601.894} C_VEL
LIN {X 0,Y 436.977,Z 419.857,A -85,B 0,C 180,E1 -9603.396,E2 -9603.396} C_VEL
LIN {X 0,Y 436.518,Z 433.354,A -85,B 0,C 180,E1 -9603.817,E2 -9603.817} C_VEL
LIN {X 0,Y 436.161,Z 446.316,A -85,B 0,C 180,E1 -9604.433,E2 -9604.433} C_VEL
LIN {X 0,Y 435.526,Z 458.124,A -85,B 0,C 180,E1 -9605.193,E2 -9605.193} C_VEL
LIN {X 0,Y 434.767,Z 469.836,A -85,B 0,C 180,E1 -9606.164,E2 -9606.164} C_VEL
LIN {X 0,Y 434.148,Z 479.239,A -85,B 0,C 180,E1 -9607.138,E2 -9607.138} C_VEL
LIN {X 0,Y 433.428,Z 488.781,A -85,B 0,C 180,E1 -9608.353,E2 -9608.353} C_VEL
LIN {X 0,Y 432.827,Z 497.961,A -85,B 0,C 180,E1 -9609.815,E2 -9609.815} C_VEL
LIN {X 0,Y 432.261,Z 505.269,A -85,B 0,C 180,E1 -9611.27,E2 -9611.27} C_VEL
LIN {X 0,Y 431.907,Z 510.164,A -85,B 0,C 180,E1 -9612.48,E2 -9612.48} C_VEL
LIN {X 0,Y 431.587,Z 515.483,A -85,B 0,C 180,E1 -9614.162,E2 -9614.162} C_VEL
LIN {X 0,Y 430.824,Z 517.4,A -85,B 0,C 180,E1 -9614.899,E2 -9614.899} C_VEL
LIN {X 0,Y 427.84,Z 520.024,A -85,B 0,C 180,E1 -9616.111,E2 -9616.111} C_VEL
LIN {X 0,Y 425.344,Z 521.572,A -85,B 0,C 180,E1 -9617.105,E2 -9617.105} C_VEL
LIN {X 0,Y 424.248,Z 522.419,A -85,B 0,C 180,E1 -9617.884,E2 -9617.884} C_VEL
LIN {X 0,Y 424.145,Z 522.61,A -85,B 0,C 180,E1 -9618.149,E2 -9618.149} C_VEL
LIN {X 0,Y 424.063,Z 523.228,A -85,B 0,C 180,E1 -9619.496,E2 -9619.496} C_VEL
LIN {X 0,Y 424.021,Z 523.181,A -85,B 0,C 180,E1 -9620.459,E2 -9620.459} C_VEL
LIN {X 0,Y 424.067,Z 522.73,A -85,B 0,C 180,E1 -9621.422,E2 -9621.422} C_VEL
LIN {X 0,Y 424.127,Z 521.842,A -85,B 0,C 180,E1 -9622.382,E2 -9622.382} C_VEL
LIN {X 0,Y 424.277,Z 520.068,A -85,B 0,C 180,E1 -9623.657,E2 -9623.657} C_VEL
LIN {X 0,Y 424.312,Z 516.751,A -85,B 0,C 180,E1 -9625.249,E2 -9625.249} C_VEL
LIN {X 0,Y 424.537,Z 512.677,A -85,B 0,C 180,E1 -9626.678,E2 -9626.678} C_VEL
LIN {X 0,Y 424.848,Z 506.449,A -85,B 0,C 180,E1 -9628.341,E2 -9628.341} C_VEL
LIN {X 0,Y 425.307,Z 499.673,A -85,B 0,C 180,E1 -9629.763,E2 -9629.763} C_VEL
LIN {X 0,Y 425.852,Z 491.238,A -85,B 0,C 180,E1 -9631.182,E2 -9631.182} C_VEL
LIN {X 0,Y 426.279,Z 482.604,A -85,B 0,C 180,E1 -9632.362,E2 -9632.362} C_VEL
LIN {X 0,Y 426.975,Z 471.954,A -85,B 0,C 180,E1 -9633.538,E2 -9633.538} C_VEL
LIN {X 0,Y 427.792,Z 461.287,A -85,B 0,C 180,E1 -9634.475,E2 -9634.475} C_VEL
LIN {X 0,Y 428.313,Z 449.419,A -85,B 0,C 180,E1 -9635.295,E2 -9635.295} C_VEL
LIN {X 0,Y 428.793,Z 437.06,A -85,B 0,C 180,E1 -9635.938,E2 -9635.938} C_VEL
LIN {X 0,Y 429.048,Z 426.133,A -85,B 0,C 180,E1 -9636.347,E2 -9636.347} C_VEL
LIN {X 0,Y 429.363,Z 412.271,A -85,B 0,C 180,E1 -9636.667,E2 -9636.667} C_VEL
LIN {X 0,Y 430.235,Z 331.134,A -85,B 0,C 180,E1 -9638.018,E2 -9638.018} C_VEL
LIN {X 0,Y 426.722,Z 312.288,A -85,B 0,C 180,E1 -9638.478,E2 -9638.478} C_VEL
LIN {X 0,Y 426.75,Z 305.356,A -85,B 0,C 180,E1 -9639.957,E2 -9639.957} C_VEL
LIN {X 0,Y 425.404,Z 297.496,A -85,B 0,C 180,E1 -9641.736,E2 -9641.736} C_VEL
LIN {X 0,Y 425.334,Z 297.499,A -85,B 0,C 180,E1 -9645.329,E2 -9645.329} C_VEL
LIN {X 0,Y 425.317,Z 297.508,A -85,B 0,C 180,E1 -9648.297,E2 -9648.297} C_VEL
LIN {X 0,Y 425.29,Z 297.504,A -85,B 0,C 180,E1 -9651.318,E2 -9651.318} C_VEL
LIN {X 0,Y 425.294,Z 297.511,A -85,B 0,C 180,E1 -9654.649,E2 -9654.649} C_VEL
LIN {X 0,Y 425.246,Z 297.51,A -85,B 0,C 180,E1 -9657.564,E2 -9657.564} C_VEL
LIN {X 0,Y 425.278,Z 297.506,A -85,B 0,C 180,E1 -9659.719,E2 -9659.719} C_VEL
LIN {X 0,Y 425.278,Z 297.51,A -85,B 0,C 180,E1 -9663.047,E2 -9663.047} C_VEL
LIN {X 0,Y 425.277,Z 297.506,A -85,B 0,C 180,E1 -9665.928,E2 -9665.928} C_VEL
LIN {X 0,Y 425.26,Z 297.515,A -85,B 0,C 180,E1 -9669.037,E2 -9669.037} C_VEL
LIN {X 0,Y 425.255,Z 297.512,A -85,B 0,C 180,E1 -9672.654,E2 -9672.654} C_VEL
LIN {X 0,Y 425.279,Z 297.511,A -85,B 0,C 180,E1 -9675.282,E2 -9675.282} C_VEL
LIN {X 0,Y 425.258,Z 297.509,A -85,B 0,C 180,E1 -9678.62,E2 -9678.62} C_VEL
LIN {X 0,Y 425.284,Z 297.511,A -85,B 0,C 180,E1 -9681.1,E2 -9681.1} C_VEL
LIN {X 0,Y 425.292,Z 297.505,A -85,B 0,C 180,E1 -9684.663,E2 -9684.663} C_VEL
LIN {X 0,Y 425.257,Z 297.509,A -85,B 0,C 180,E1 -9688.072,E2 -9688.072} C_VEL
LIN {X 0,Y 425.323,Z 297.506,A -85,B 0,C 180,E1 -9691.367,E2 -9691.367} C_VEL
LIN {X 0,Y 425.276,Z 297.506,A -85,B 0,C 180,E1 -9694.553,E2 -9694.553} C_VEL
LIN {X 0,Y 425.276,Z 297.506,A -85,B 0,C 180,E1 -9696.633,E2 -9696.633} C_VEL
LIN {X 0,Y 425.287,Z 297.512,A -85,B 0,C 180,E1 -9699.694,E2 -9699.694} C_VEL
LIN {X 0,Y 425.335,Z 297.499,A -85,B 0,C 180,E1 -9702.697,E2 -9702.697} C_VEL
LIN {X 0,Y 425.341,Z 297.502,A -85,B 0,C 180,E1 -9705.65,E2 -9705.65} C_VEL
LIN {X 0,Y 425.342,Z 297.499,A -85,B 0,C 180,E1 -9708.564,E2 -9708.564} C_VEL
LIN {X 0,Y 425.428,Z 297.488,A -85,B 0,C 180,E1 -9711.45,E2 -9711.45} C_VEL
LIN {X 0,Y 425.532,Z 297.48,A -85,B 0,C 180,E1 -9714.313,E2 -9714.313} C_VEL
LIN {X 0,Y 425.565,Z 297.476,A -85,B 0,C 180,E1 -9718.107,E2 -9718.107} C_VEL
LIN {X 0,Y 425.692,Z 297.458,A -85,B 0,C 180,E1 -9720,E2 -9720} C_VEL
LIN {X 0,Y 425.537,Z 297.476,A -85,B 0,C 180,E1 -9722.84,E2 -9722.84} C_VEL
LIN {X 0,Y 425.521,Z 297.481,A -85,B 0,C 180,E1 -9726.639,E2 -9726.639} C_VEL
LIN {X 0,Y 425.394,Z 297.491,A -85,B 0,C 180,E1 -9729.51,E2 -9729.51} C_VEL
LIN {X 0,Y 425.385,Z 297.497,A -85,B 0,C 180,E1 -9732.904,E2 -9732.904} C_VEL
LIN {X 0,Y 425.353,Z 297.502,A -85,B 0,C 180,E1 -9736.605,E2 -9736.605} C_VEL
LIN {X 0,Y 425.321,Z 297.501,A -85,B 0,C 180,E1 -9739.636,E2 -9739.636} C_VEL
LIN {X 0,Y 425.3,Z 297.506,A -85,B 0,C 180,E1 -9743.366,E2 -9743.366} C_VEL
LIN {X 0,Y 425.342,Z 297.503,A -85,B 0,C 180,E1 -9746.845,E2 -9746.845} C_VEL
LIN {X 0,Y 425.313,Z 297.503,A -85,B 0,C 180,E1 -9749.718,E2 -9749.718} C_VEL
LIN {X 0,Y 425.279,Z 297.512,A -85,B 0,C 180,E1 -9753.049,E2 -9753.049} C_VEL
LIN {X 0,Y 425.279,Z 297.507,A -85,B 0,C 180,E1 -9755.93,E2 -9755.93} C_VEL
LIN {X 0,Y 425.298,Z 297.507,A -85,B 0,C 180,E1 -9759.045,E2 -9759.045} C_VEL
LIN {X 0,Y 425.274,Z 297.506,A -85,B 0,C 180,E1 -9762.653,E2 -9762.653} C_VEL
LIN {X 0,Y 425.257,Z 297.51,A -85,B 0,C 180,E1 -9766.045,E2 -9766.045} C_VEL
LIN {X 0,Y 425.27,Z 297.507,A -85,B 0,C 180,E1 -9768.622,E2 -9768.622} C_VEL
LIN {X 0,Y 425.294,Z 297.505,A -85,B 0,C 180,E1 -9771.102,E2 -9771.102} C_VEL
LIN {X 0,Y 425.297,Z 297.503,A -85,B 0,C 180,E1 -9774.665,E2 -9774.665} C_VEL
LIN {X 0,Y 425.263,Z 297.513,A -85,B 0,C 180,E1 -9778.074,E2 -9778.074} C_VEL
LIN {X 0,Y 425.33,Z 297.505,A -85,B 0,C 180,E1 -9781.369,E2 -9781.369} C_VEL
LIN {X 0,Y 425.415,Z 297.559,A -85,B 0,C 180,E1 -9782.939,E2 -9782.939} C_VEL
LIN {X 0,Y 427.958,Z 311.378,A -85,B 0,C 180,E1 -9785.761,E2 -9785.761} C_VEL
LIN {X 0,Y 427.289,Z 324.677,A -85,B 0,C 180,E1 -9788.28,E2 -9788.28} C_VEL
LIN {X 0,Y 426.327,Z 341.992,A -85,B 0,C 180,E1 -9791.522,E2 -9791.522} C_VEL
LIN {X 0,Y 429.968,Z 368.2,A -85,B 0,C 180,E1 -9792.112,E2 -9792.112} C_VEL
LIN {X 0,Y 429.107,Z 450.323,A -85,B 0,C 180,E1 -9793.498,E2 -9793.498} C_VEL
LIN {X 0,Y 428.656,Z 463.688,A -85,B 0,C 180,E1 -9793.908,E2 -9793.908} C_VEL
LIN {X 0,Y 428.139,Z 475.923,A -85,B 0,C 180,E1 -9794.469,E2 -9794.469} C_VEL
LIN {X 0,Y 427.475,Z 488.248,A -85,B 0,C 180,E1 -9795.237,E2 -9795.237} C_VEL
LIN {X 0,Y 426.815,Z 499.467,A -85,B 0,C 180,E1 -9796.147,E2 -9796.147} C_VEL
LIN {X 0,Y 426.148,Z 510.382,A -85,B 0,C 180,E1 -9797.258,E2 -9797.258} C_VEL
LIN {X 0,Y 425.634,Z 518.949,A -85,B 0,C 180,E1 -9798.331,E2 -9798.331} C_VEL
LIN {X 0,Y 425.011,Z 528.214,A -85,B 0,C 180,E1 -9799.761,E2 -9799.761} C_VEL
LIN {X 0,Y 424.657,Z 535.666,A -85,B 0,C 180,E1 -9801.195,E2 -9801.195} C_VEL
LIN {X 0,Y 424.341,Z 542.508,A -85,B 0,C 180,E1 -9802.865,E2 -9802.865} C_VEL
LIN {X 0,Y 424.183,Z 547.013,A -85,B 0,C 180,E1 -9804.295,E2 -9804.295} C_VEL
LIN {X 0,Y 424.199,Z 549.391,A -85,B 0,C 180,E1 -9805.249,E2 -9805.249} C_VEL
LIN {X 0,Y 424.102,Z 551.328,A -85,B 0,C 180,E1 -9806.2,E2 -9806.2} C_VEL
LIN {X 0,Y 424.164,Z 552.844,A -85,B 0,C 180,E1 -9807.151,E2 -9807.151} C_VEL
LIN {X 0,Y 424.145,Z 553.902,A -85,B 0,C 180,E1 -9808.101,E2 -9808.101} C_VEL
LIN {X 0,Y 424.108,Z 554.842,A -85,B 0,C 180,E1 -9810.001,E2 -9810.001} C_VEL
LIN {X 0,Y 424.091,Z 554.725,A -85,B 0,C 180,E1 -9810.95,E2 -9810.95} C_VEL
LIN {X 0,Y 424.143,Z 554.176,A -85,B 0,C 180,E1 -9811.9,E2 -9811.9} C_VEL
LIN {X 0,Y 424.133,Z 553.232,A -85,B 0,C 180,E1 -9812.85,E2 -9812.85} C_VEL
LIN {X 0,Y 424.1,Z 551.893,A -85,B 0,C 180,E1 -9813.801,E2 -9813.801} C_VEL
LIN {X 0,Y 424.207,Z 549.071,A -85,B 0,C 180,E1 -9815.229,E2 -9815.229} C_VEL
LIN {X 0,Y 424.3,Z 545.229,A -85,B 0,C 180,E1 -9816.659,E2 -9816.659} C_VEL
LIN {X 0,Y 424.523,Z 540.271,A -85,B 0,C 180,E1 -9818.09,E2 -9818.09} C_VEL
LIN {X 0,Y 424.872,Z 534.051,A -85,B 0,C 180,E1 -9819.522,E2 -9819.522} C_VEL
LIN {X 0,Y 425.404,Z 526.313,A -85,B 0,C 180,E1 -9820.952,E2 -9820.952} C_VEL
LIN {X 0,Y 426.19,Z 516.637,A -85,B 0,C 180,E1 -9822.379,E2 -9822.379} C_VEL
LIN {X 0,Y 426.883,Z 506.68,A -85,B 0,C 180,E1 -9823.568,E2 -9823.568} C_VEL
LIN {X 0,Y 427.562,Z 496.849,A -85,B 0,C 180,E1 -9824.517,E2 -9824.517} C_VEL
LIN {X 0,Y 428.422,Z 484.437,A -85,B 0,C 180,E1 -9825.461,E2 -9825.461} C_VEL
LIN {X 0,Y 429.192,Z 472.271,A -85,B 0,C 180,E1 -9826.163,E2 -9826.163} C_VEL
LIN {X 0,Y 429.78,Z 459.561,A -85,B 0,C 180,E1 -9826.69,E2 -9826.69} C_VEL
LIN {X 0,Y 430.2,Z 446.188,A -85,B 0,C 180,E1 -9827.04,E2 -9827.04} C_VEL
LIN {X 0,Y 431.041,Z 367.108,A -85,B 0,C 180,E1 -9828.385,E2 -9828.385} C_VEL
LIN {X 0,Y 427.644,Z 346.09,A -85,B 0,C 180,E1 -9828.928,E2 -9828.928} C_VEL
LIN {X 0,Y 426.803,Z 341.677,A -85,B 0,C 180,E1 -9829.055,E2 -9829.055} C_VEL
LIN {X 0,Y 427.952,Z 323.91,A -85,B 0,C 180,E1 -9832.444,E2 -9832.444} C_VEL
LIN {X 0,Y 428.573,Z 313.513,A -85,B 0,C 180,E1 -9834.461,E2 -9834.461} C_VEL
LIN {X 0,Y 426.663,Z 303.279,A -85,B 0,C 180,E1 -9836.64,E2 -9836.64} C_VEL
LIN {X 0,Y 425.381,Z 297.504,A -85,B 0,C 180,E1 -9837.957,E2 -9837.957} C_VEL
LIN {X 0,Y 425.29,Z 297.51,A -85,B 0,C 180,E1 -9840.816,E2 -9840.816} C_VEL
LIN {X 0,Y 425.313,Z 297.511,A -85,B 0,C 180,E1 -9844.288,E2 -9844.288} C_VEL
LIN {X 0,Y 425.28,Z 297.509,A -85,B 0,C 180,E1 -9847.694,E2 -9847.694} C_VEL
LIN {X 0,Y 425.281,Z 297.512,A -85,B 0,C 180,E1 -9850.52,E2 -9850.52} C_VEL
LIN {X 0,Y 425.258,Z 297.511,A -85,B 0,C 180,E1 -9853.351,E2 -9853.351} C_VEL
LIN {X 0,Y 425.258,Z 297.514,A -85,B 0,C 180,E1 -9856.649,E2 -9856.649} C_VEL
LIN {X 0,Y 425.286,Z 297.503,A -85,B 0,C 180,E1 -9859.872,E2 -9859.872} C_VEL
LIN {X 0,Y 425.278,Z 297.51,A -85,B 0,C 180,E1 -9862.488,E2 -9862.488} C_VEL
LIN {X 0,Y 425.307,Z 297.499,A -85,B 0,C 180,E1 -9865.817,E2 -9865.817} C_VEL
LIN {X 0,Y 425.29,Z 297.506,A -85,B 0,C 180,E1 -9869.239,E2 -9869.239} C_VEL
LIN {X 0,Y 425.348,Z 297.498,A -85,B 0,C 180,E1 -9872.442,E2 -9872.442} C_VEL
LIN {X 0,Y 425.349,Z 297.5,A -85,B 0,C 180,E1 -9875.602,E2 -9875.602} C_VEL
LIN {X 0,Y 425.292,Z 297.505,A -85,B 0,C 180,E1 -9878.681,E2 -9878.681} C_VEL
LIN {X 0,Y 425.332,Z 297.502,A -85,B 0,C 180,E1 -9881.703,E2 -9881.703} C_VEL
LIN {X 0,Y 425.348,Z 297.496,A -85,B 0,C 180,E1 -9884.67,E2 -9884.67} C_VEL
LIN {X 0,Y 425.411,Z 297.495,A -85,B 0,C 180,E1 -9887.598,E2 -9887.598} C_VEL
LIN {X 0,Y 425.441,Z 297.485,A -85,B 0,C 180,E1 -9891.45,E2 -9891.45} C_VEL
LIN {X 0,Y 425.552,Z 297.467,A -85,B 0,C 180,E1 -9894.313,E2 -9894.313} C_VEL
LIN {X 0,Y 425.571,Z 297.467,A -85,B 0,C 180,E1 -9898.107,E2 -9898.107} C_VEL
LIN {X 0,Y 425.7,Z 297.453,A -85,B 0,C 180,E1 -9900,E2 -9900} C_VEL
LIN {X 0,Y 425.544,Z 297.467,A -85,B 0,C 180,E1 -9902.84,E2 -9902.84} C_VEL
LIN {X 0,Y 425.526,Z 297.474,A -85,B 0,C 180,E1 -9906.639,E2 -9906.639} C_VEL
LIN {X 0,Y 425.399,Z 297.49,A -85,B 0,C 180,E1 -9909.509,E2 -9909.509} C_VEL
LIN {X 0,Y 425.392,Z 297.493,A -85,B 0,C 180,E1 -9912.904,E2 -9912.904} C_VEL
LIN {X 0,Y 425.36,Z 297.498,A -85,B 0,C 180,E1 -9916.605,E2 -9916.605} C_VEL
LIN {X 0,Y 425.327,Z 297.5,A -85,B 0,C 180,E1 -9919.636,E2 -9919.636} C_VEL
LIN {X 0,Y 425.287,Z 297.507,A -85,B 0,C 180,E1 -9922.339,E2 -9922.339} C_VEL
LIN {X 0,Y 425.294,Z 297.504,A -85,B 0,C 180,E1 -9925.445,E2 -9925.445} C_VEL
LIN {X 0,Y 425.33,Z 297.5,A -85,B 0,C 180,E1 -9928.632,E2 -9928.632} C_VEL
LIN {X 0,Y 425.263,Z 297.505,A -85,B 0,C 180,E1 -9931.927,E2 -9931.927} C_VEL
LIN {X 0,Y 425.298,Z 297.508,A -85,B 0,C 180,E1 -9935.336,E2 -9935.336} C_VEL
LIN {X 0,Y 425.301,Z 297.507,A -85,B 0,C 180,E1 -9938.898,E2 -9938.898} C_VEL
LIN {X 0,Y 425.289,Z 297.506,A -85,B 0,C 180,E1 -9941.958,E2 -9941.958} C_VEL
LIN {X 0,Y 425.284,Z 297.51,A -85,B 0,C 180,E1 -9945.283,E2 -9945.283} C_VEL
LIN {X 0,Y 425.274,Z 297.508,A -85,B 0,C 180,E1 -9948.621,E2 -9948.621} C_VEL
LIN {X 0,Y 425.297,Z 297.509,A -85,B 0,C 180,E1 -9951.101,E2 -9951.101} C_VEL
LIN {X 0,Y 425.3,Z 297.504,A -85,B 0,C 180,E1 -9954.664,E2 -9954.664} C_VEL
LIN {X 0,Y 425.325,Z 297.65,A -85,B 0,C 180,E1 -9957.692,E2 -9957.692} C_VEL
LIN {X 0,Y 427.243,Z 307.139,A -85,B 0,C 180,E1 -9959.886,E2 -9959.886} C_VEL
LIN {X 0,Y 427.185,Z 312.364,A -85,B 0,C 180,E1 -9961.005,E2 -9961.005} C_VEL
LIN {X 0,Y 431.41,Z 331.365,A -85,B 0,C 180,E1 -9961.567,E2 -9961.567} C_VEL
LIN {X 0,Y 430.286,Z 419.769,A -85,B 0,C 180,E1 -9963.08,E2 -9963.08} C_VEL
LIN {X 0,Y 429.812,Z 433.381,A -85,B 0,C 180,E1 -9963.507,E2 -9963.507} C_VEL
LIN {X 0,Y 429.415,Z 446.487,A -85,B 0,C 180,E1 -9964.137,E2 -9964.137} C_VEL
LIN {X 0,Y 428.759,Z 458.26,A -85,B 0,C 180,E1 -9964.904,E2 -9964.904} C_VEL
LIN {X 0,Y 427.963,Z 469.993,A -85,B 0,C 180,E1 -9965.889,E2 -9965.889} C_VEL
LIN {X 0,Y 427.205,Z 480.606,A -85,B 0,C 180,E1 -9967.018,E2 -9967.018} C_VEL
LIN {X 0,Y 426.47,Z 489.808,A -85,B 0,C 180,E1 -9968.236,E2 -9968.236} C_VEL
LIN {X 0,Y 425.84,Z 498.855,A -85,B 0,C 180,E1 -9969.721,E2 -9969.721} C_VEL
LIN {X 0,Y 425.233,Z 506.001,A -85,B 0,C 180,E1 -9971.199,E2 -9971.199} C_VEL
LIN {X 0,Y 424.82,Z 511.662,A -85,B 0,C 180,E1 -9972.675,E2 -9972.675} C_VEL
LIN {X 0,Y 424.509,Z 516.186,A -85,B 0,C 180,E1 -9974.195,E2 -9974.195} C_VEL
LIN {X 0,Y 424.276,Z 519.342,A -85,B 0,C 180,E1 -9975.613,E2 -9975.613} C_VEL
LIN {X 0,Y 424.173,Z 520.957,A -85,B 0,C 180,E1 -9976.587,E2 -9976.587} C_VEL
LIN {X 0,Y 424.145,Z 522.61,A -85,B 0,C 180,E1 -9978.149,E2 -9978.149} C_VEL
LIN {X 0,Y 423.43,Z 523.117,A -85,B 0,C 180,E1 -9978.939,E2 -9978.939} C_VEL
LIN {X 0,Y 420.531,Z 523.448,A -85,B 0,C 180,E1 -9980.227,E2 -9980.227} C_VEL
LIN {X 0,Y 418.123,Z 523.14,A -85,B 0,C 180,E1 -9981.264,E2 -9981.264} C_VEL
LIN {X 0,Y 417.113,Z 522.478,A -85,B 0,C 180,E1 -9982.061,E2 -9982.061} C_VEL
LIN {X 0,Y 417.042,Z 522.162,A -85,B 0,C 180,E1 -9982.329,E2 -9982.329} C_VEL
LIN {X 0,Y 417.214,Z 519.386,A -85,B 0,C 180,E1 -9984.199,E2 -9984.199} C_VEL
LIN {X 0,Y 417.253,Z 516.115,A -85,B 0,C 180,E1 -9985.653,E2 -9985.653} C_VEL
LIN {X 0,Y 417.529,Z 511.77,A -85,B 0,C 180,E1 -9987.105,E2 -9987.105} C_VEL
LIN {X 0,Y 417.828,Z 506.253,A -85,B 0,C 180,E1 -9988.554,E2 -9988.554} C_VEL
LIN {X 0,Y 418.313,Z 499.37,A -85,B 0,C 180,E1 -9989.999,E2 -9989.999} C_VEL
LIN {X 0,Y 418.903,Z 490.755,A -85,B 0,C 180,E1 -9991.442,E2 -9991.442} C_VEL
LIN {X 0,Y 419.355,Z 481.973,A -85,B 0,C 180,E1 -9992.641,E2 -9992.641} C_VEL
LIN {X 0,Y 420.019,Z 472.302,A -85,B 0,C 180,E1 -9993.717,E2 -9993.717} C_VEL
LIN {X 0,Y 420.866,Z 461.657,A -85,B 0,C 180,E1 -9994.669,E2 -9994.669} C_VEL
LIN {X 0,Y 421.406,Z 449.819,A -85,B 0,C 180,E1 -9995.502,E2 -9995.502} C_VEL
LIN {X 0,Y 421.898,Z 437.501,A -85,B 0,C 180,E1 -9996.155,E2 -9996.155} C_VEL
LIN {X 0,Y 422.145,Z 426.657,A -85,B 0,C 180,E1 -9996.572,E2 -9996.572} C_VEL
LIN {X 0,Y 422.492,Z 413.016,A -85,B 0,C 180,E1 -9996.896,E2 -9996.896} C_VEL
LIN {X 0,Y 423.27,Z 331.436,A -85,B 0,C 180,E1 -9998.281,E2 -9998.281} C_VEL
LIN {X 0,Y 419.774,Z 312.456,A -85,B 0,C 180,E1 -9998.766,E2 -9998.766} C_VEL
LIN {X 0,Y 419.713,Z 306.193,A -85,B 0,C 180,E1 -10000.126,E2 -10000.126} C_VEL
LIN {X 0,Y 418.394,Z 298.37,A -85,B 0,C 180,E1 -10001.935,E2 -10001.935} C_VEL
LIN {X 0,Y 418.29,Z 298.377,A -85,B 0,C 180,E1 -10005.594,E2 -10005.594} C_VEL
LIN {X 0,Y 418.272,Z 298.384,A -85,B 0,C 180,E1 -10008.617,E2 -10008.617} C_VEL
LIN {X 0,Y 418.231,Z 298.384,A -85,B 0,C 180,E1 -10011.696,E2 -10011.696} C_VEL
LIN {X 0,Y 418.241,Z 298.387,A -85,B 0,C 180,E1 -10014.852,E2 -10014.852} C_VEL
LIN {X 0,Y 418.209,Z 298.388,A -85,B 0,C 180,E1 -10018.068,E2 -10018.068} C_VEL
LIN {X 0,Y 418.235,Z 298.387,A -85,B 0,C 180,E1 -10021.018,E2 -10021.018} C_VEL
LIN {X 0,Y 418.243,Z 298.382,A -85,B 0,C 180,E1 -10023.676,E2 -10023.676} C_VEL
LIN {X 0,Y 418.234,Z 298.387,A -85,B 0,C 180,E1 -10027.223,E2 -10027.223} C_VEL
LIN {X 0,Y 418.206,Z 298.393,A -85,B 0,C 180,E1 -10030.867,E2 -10030.867} C_VEL
LIN {X 0,Y 418.198,Z 298.389,A -85,B 0,C 180,E1 -10033.728,E2 -10033.728} C_VEL
LIN {X 0,Y 418.2,Z 298.388,A -85,B 0,C 180,E1 -10036.448,E2 -10036.448} C_VEL
LIN {X 0,Y 418.21,Z 298.393,A -85,B 0,C 180,E1 -10039.131,E2 -10039.131} C_VEL
LIN {X 0,Y 418.217,Z 298.385,A -85,B 0,C 180,E1 -10042.167,E2 -10042.167} C_VEL
LIN {X 0,Y 418.258,Z 298.388,A -85,B 0,C 180,E1 -10045.419,E2 -10045.419} C_VEL
LIN {X 0,Y 418.203,Z 298.387,A -85,B 0,C 180,E1 -10048.603,E2 -10048.603} C_VEL
LIN {X 0,Y 418.282,Z 298.38,A -85,B 0,C 180,E1 -10051.936,E2 -10051.936} C_VEL
LIN {X 0,Y 418.264,Z 298.382,A -85,B 0,C 180,E1 -10055.161,E2 -10055.161} C_VEL
LIN {X 0,Y 418.225,Z 298.386,A -85,B 0,C 180,E1 -10058.303,E2 -10058.303} C_VEL
LIN {X 0,Y 418.275,Z 298.381,A -85,B 0,C 180,E1 -10061.383,E2 -10061.383} C_VEL
LIN {X 0,Y 418.302,Z 298.377,A -85,B 0,C 180,E1 -10064.406,E2 -10064.406} C_VEL
LIN {X 0,Y 418.347,Z 298.37,A -85,B 0,C 180,E1 -10067.385,E2 -10067.385} C_VEL
LIN {X 0,Y 418.332,Z 298.375,A -85,B 0,C 180,E1 -10070.329,E2 -10070.329} C_VEL
LIN {X 0,Y 418.45,Z 298.356,A -85,B 0,C 180,E1 -10073.248,E2 -10073.248} C_VEL
LIN {X 0,Y 418.328,Z 298.371,A -85,B 0,C 180,E1 -10075.182,E2 -10075.182} C_VEL
LIN {X 0,Y 418.534,Z 298.351,A -85,B 0,C 180,E1 -10078.076,E2 -10078.076} C_VEL
LIN {X 0,Y 418.661,Z 298.334,A -85,B 0,C 180,E1 -10080,E2 -10080} C_VEL
LIN {X 0,Y 418.493,Z 298.353,A -85,B 0,C 180,E1 -10082.888,E2 -10082.888} C_VEL
LIN {X 0,Y 418.484,Z 298.357,A -85,B 0,C 180,E1 -10086.751,E2 -10086.751} C_VEL
LIN {X 0,Y 418.334,Z 298.371,A -85,B 0,C 180,E1 -10089.672,E2 -10089.672} C_VEL
LIN {X 0,Y 418.338,Z 298.374,A -85,B 0,C 180,E1 -10093.001,E2 -10093.001} C_VEL
LIN {X 0,Y 418.305,Z 298.382,A -85,B 0,C 180,E1 -10096.736,E2 -10096.736} C_VEL
LIN {X 0,Y 418.263,Z 298.379,A -85,B 0,C 180,E1 -10099.791,E2 -10099.791} C_VEL
LIN {X 0,Y 418.231,Z 298.389,A -85,B 0,C 180,E1 -10102.737,E2 -10102.737} C_VEL
LIN {X 0,Y 418.264,Z 298.379,A -85,B 0,C 180,E1 -10105.905,E2 -10105.905} C_VEL
LIN {X 0,Y 418.269,Z 298.386,A -85,B 0,C 180,E1 -10109.162,E2 -10109.162} C_VEL
LIN {X 0,Y 418.255,Z 298.384,A -85,B 0,C 180,E1 -10112.845,E2 -10112.845} C_VEL
LIN {X 0,Y 418.243,Z 298.382,A -85,B 0,C 180,E1 -10116.239,E2 -10116.239} C_VEL
LIN {X 0,Y 418.25,Z 298.385,A -85,B 0,C 180,E1 -10119.682,E2 -10119.682} C_VEL
LIN {X 0,Y 418.228,Z 298.384,A -85,B 0,C 180,E1 -10122.322,E2 -10122.322} C_VEL
LIN {X 0,Y 418.234,Z 298.386,A -85,B 0,C 180,E1 -10125.11,E2 -10125.11} C_VEL
LIN {X 0,Y 418.236,Z 298.388,A -85,B 0,C 180,E1 -10127.768,E2 -10127.768} C_VEL
LIN {X 0,Y 418.242,Z 298.382,A -85,B 0,C 180,E1 -10130.622,E2 -10130.622} C_VEL
LIN {X 0,Y 418.24,Z 298.387,A -85,B 0,C 180,E1 -10133.977,E2 -10133.977} C_VEL
LIN {X 0,Y 418.256,Z 298.381,A -85,B 0,C 180,E1 -10137.157,E2 -10137.157} C_VEL
LIN {X 0,Y 418.267,Z 298.383,A -85,B 0,C 180,E1 -10140.896,E2 -10140.896} C_VEL
LIN {X 0,Y 418.369,Z 298.484,A -85,B 0,C 180,E1 -10142.742,E2 -10142.742} C_VEL
